C07276=1031.156,417.166,352.413,174.368,47.663,159.722
C07277=1031.145,416.920,352.461,174.356,47.658,159.719
C07278=1031.134,416.675,352.508,174.343,47.654,159.716
C07279=1031.123,416.430,352.556,174.331,47.649,159.713
C07280=1031.112,416.185,352.603,174.319,47.645,159.710
C07281=1031.101,415.939,352.650,174.306,47.640,159.707
C07282=1031.090,415.694,352.698,174.294,47.636,159.704
C07283=1031.079,415.449,352.745,174.282,47.631,159.701
C07284=1031.068,415.203,352.792,174.270,47.627,159.698
C07285=1031.057,414.958,352.839,174.258,47.622,159.696
C07286=1031.046,414.713,352.887,174.246,47.618,159.693
C07287=1031.035,414.468,352.934,174.234,47.614,159.690
C07288=1031.025,414.222,352.981,174.222,47.610,159.687
C07289=1031.014,413.977,353.028,174.210,47.605,159.684
C07290=1031.003,413.731,353.075,174.198,47.601,159.681
C07291=1030.992,413.486,353.122,174.186,47.597,159.679
C07292=1030.981,413.241,353.169,174.174,47.592,159.676
C07293=1030.970,412.995,353.216,174.162,47.588,159.673
C07294=1030.960,412.750,353.262,174.151,47.584,159.671
C07295=1030.950,412.505,353.309,174.139,47.579,159.668
C07296=1030.939,412.260,353.356,174.127,47.576,159.665
C07297=1030.928,412.014,353.403,174.115,47.571,159.662
C07298=1030.917,411.768,353.449,174.104,47.567,159.660
C07299=1030.906,411.523,353.496,174.093,47.563,159.657
C07300=1030.896,411.278,353.543,174.081,47.558,159.654
C07301=1030.885,411.032,353.589,174.070,47.554,159.652
C07302=1030.875,410.787,353.636,174.058,47.550,159.649
C07303=1030.865,410.541,353.682,174.046,47.546,159.646
C07304=1030.854,410.296,353.728,174.035,47.542,159.644
C07305=1030.843,410.051,353.775,174.024,47.538,159.641
C07306=1030.833,409.805,353.821,174.013,47.534,159.638
C07307=1030.823,409.559,353.867,174.001,47.530,159.636
C07308=1030.812,409.314,353.913,173.990,47.526,159.633
C07309=1030.800,409.049,353.962,173.978,47.522,159.630
C07310=1030.789,408.784,354.012,173.966,47.518,159.628
C07311=1030.778,408.520,354.062,173.953,47.513,159.625
C07312=1030.766,408.256,354.111,173.942,47.509,159.622
C07313=1030.756,408.010,354.158,173.930,47.505,159.620
C07314=1030.746,407.764,354.204,173.919,47.501,159.617
C07315=1030.735,407.518,354.249,173.908,47.498,159.615
C07316=1030.725,407.272,354.295,173.897,47.494,159.612
C07317=1030.715,407.028,354.340,173.886,47.490,159.610
C07318=1030.704,406.782,354.386,173.875,47.486,159.607
C07319=1030.693,406.536,354.432,173.864,47.482,159.605
C07320=1030.684,406.291,354.477,173.853,47.478,159.602
C07321=1030.673,406.045,354.523,173.843,47.475,159.600
C07322=1030.663,405.800,354.569,173.831,47.471,159.597
C07323=1030.653,405.554,354.613,173.821,47.467,159.595
C07324=1030.643,405.308,354.660,173.810,47.463,159.592
C07325=1030.633,405.062,354.705,173.799,47.460,159.590
C07326=1030.623,404.817,354.751,173.788,47.456,159.587
C07327=1030.612,404.571,354.796,173.778,47.452,159.585
C07328=1030.602,404.326,354.841,173.768,47.449,159.583
C07329=1030.593,404.080,354.886,173.756,47.445,159.580
C07330=1030.582,403.834,354.931,173.746,47.441,159.578
C07331=1030.572,403.589,354.977,173.735,47.438,159.575
C07332=1030.562,403.343,355.022,173.725,47.434,159.573
C07333=1030.552,403.098,355.067,173.714,47.430,159.571
C07334=1030.542,402.852,355.112,173.703,47.427,159.568
C07335=1030.532,402.606,355.157,173.693,47.423,159.566
C07336=1030.522,402.361,355.203,173.683,47.419,159.564
C07337=1030.512,402.116,355.247,173.673,47.416,159.561
C07338=1030.502,401.869,355.293,173.662,47.413,159.559
C07339=1030.492,401.624,355.337,173.651,47.409,159.557
C07340=1030.483,401.378,355.382,173.641,47.406,159.555
C07341=1030.473,401.131,355.427,173.631,47.402,159.552
C07342=1030.463,400.886,355.472,173.620,47.399,159.550
C07343=1030.453,400.640,355.516,173.610,47.395,159.548
C07344=1030.443,400.395,355.561,173.600,47.392,159.545
C07345=1030.433,400.150,355.605,173.590,47.388,159.543
C07346=1030.424,399.904,355.650,173.580,47.385,159.541
C07347=1030.413,399.657,355.695,173.570,47.382,159.539
C07348=1030.404,399.411,355.739,173.559,47.378,159.536
C07349=1030.394,399.166,355.784,173.549,47.375,159.534
C07350=1030.384,398.920,355.828,173.539,47.372,159.532
C07351=1030.374,398.674,355.872,173.529,47.369,159.530
C07352=1030.365,398.428,355.916,173.519,47.365,159.528
C07353=1030.354,398.183,355.960,173.509,47.361,159.525
C07354=1030.345,397.937,356.004,173.499,47.358,159.523
C07355=1030.336,397.691,356.049,173.489,47.355,159.521
C07356=1030.325,397.446,356.093,173.479,47.352,159.519
C07357=1030.316,397.199,356.137,173.469,47.349,159.517
C07358=1030.306,396.953,356.181,173.460,47.346,159.515
C07359=1030.296,396.707,356.225,173.450,47.343,159.513
C07360=1030.287,396.462,356.269,173.440,47.339,159.510
C07361=1030.278,396.217,356.313,173.430,47.336,159.508
C07362=1030.268,395.971,356.357,173.420,47.333,159.506
C07363=1030.258,395.725,356.401,173.410,47.330,159.504
C07364=1030.248,395.479,356.444,173.401,47.327,159.502
C07365=1030.239,395.233,356.488,173.391,47.324,159.500
C07366=1030.229,394.989,356.532,173.381,47.320,159.498
C07367=1030.220,394.744,356.575,173.373,47.317,159.496
C07368=1030.211,394.500,356.618,173.363,47.314,159.494
C07369=1030.201,394.255,356.662,173.353,47.312,159.492
C07370=1030.192,394.011,356.705,173.343,47.308,159.490
C07371=1030.182,393.766,356.748,173.334,47.306,159.488
C07372=1030.173,393.521,356.791,173.325,47.303,159.486
C07373=1030.164,393.275,356.835,173.315,47.299,159.484
C07374=1030.154,393.030,356.879,173.306,47.297,159.482
C07375=1030.144,392.783,356.921,173.296,47.294,159.480
C07376=1030.135,392.538,356.965,173.286,47.291,159.478
C07377=1030.125,392.291,357.008,173.278,47.288,159.476
C07378=1030.116,392.046,357.052,173.268,47.285,159.474
C07379=1030.107,391.799,357.095,173.258,47.282,159.472
C07380=1030.098,391.554,357.138,173.249,47.279,159.470
C07381=1030.088,391.308,357.181,173.240,47.276,159.468
C07382=1030.079,391.061,357.224,173.230,47.273,159.466
C07383=1030.069,390.816,357.268,173.221,47.271,159.464
C07384=1030.060,390.570,357.310,173.212,47.268,159.462
C07385=1030.051,390.323,357.353,173.203,47.265,159.460
C07386=1030.042,390.077,357.396,173.193,47.262,159.458
C07387=1030.032,389.831,357.440,173.185,47.259,159.456
C07388=1030.023,389.586,357.482,173.175,47.256,159.454
C07389=1030.013,389.339,357.525,173.166,47.254,159.452
C07390=1030.005,389.093,357.568,173.157,47.251,159.451
C07391=1029.995,388.847,357.611,173.148,47.249,159.449
C07392=1029.986,388.601,357.653,173.139,47.245,159.447
C07393=1029.976,388.355,357.696,173.130,47.243,159.445
C07394=1029.968,388.108,357.738,173.120,47.241,159.443
C07395=1029.958,387.862,357.781,173.112,47.238,159.441
C07396=1029.949,387.616,357.823,173.102,47.235,159.439
C07397=1029.941,387.370,357.866,173.094,47.232,159.438
C07398=1029.931,387.124,357.909,173.085,47.230,159.436
C07399=1029.921,386.878,357.952,173.076,47.227,159.434
C07400=1029.913,386.632,357.993,173.067,47.225,159.432
C07401=1029.903,386.386,358.036,173.059,47.222,159.430
C07402=1029.894,386.139,358.078,173.049,47.219,159.428
C07403=1029.885,385.893,358.120,173.041,47.217,159.427
C07404=1029.876,385.647,358.162,173.032,47.215,159.425
C07405=1029.866,385.401,358.204,173.023,47.212,159.423
C07406=1029.857,385.155,358.246,173.014,47.210,159.421
C07407=1029.848,384.909,358.289,173.006,47.207,159.420
C07408=1029.839,384.662,358.331,172.997,47.205,159.418
C07409=1029.830,384.415,358.372,172.988,47.202,159.416
C07410=1029.820,384.170,358.415,172.980,47.199,159.414
C07411=1029.812,383.923,358.457,172.970,47.197,159.412
C07412=1029.803,383.677,358.498,172.962,47.195,159.411
C07413=1029.794,383.431,358.540,172.954,47.192,159.409
C07414=1029.784,383.185,358.582,172.945,47.190,159.407
C07415=1029.776,382.938,358.625,172.936,47.188,159.406
C07416=1029.767,382.692,358.666,172.928,47.185,159.404
C07417=1029.758,382.445,358.708,172.919,47.183,159.402
C07418=1029.749,382.199,358.750,172.911,47.181,159.401
C07419=1029.741,381.953,358.792,172.902,47.178,159.399
C07420=1029.732,381.706,358.833,172.893,47.176,159.397
C07421=1029.723,381.460,358.875,172.885,47.174,159.395
C07422=1029.714,381.214,358.917,172.877,47.171,159.394
C07423=1029.705,380.968,358.958,172.868,47.169,159.392
C07424=1029.696,380.722,359.000,172.860,47.167,159.390
C07425=1029.688,380.495,359.038,172.852,47.165,159.389
C07426=1029.679,380.268,359.076,172.845,47.162,159.387
C07427=1029.672,380.041,359.114,172.837,47.160,159.386
C07428=1029.663,379.814,359.153,172.829,47.159,159.384
C07429=1029.656,379.587,359.191,172.822,47.156,159.383
C07430=1029.648,379.361,359.229,172.814,47.155,159.381
C07431=1029.639,379.133,359.267,172.806,47.153,159.380
C07432=1029.631,378.907,359.306,172.799,47.150,159.378
C07433=1029.623,378.660,359.347,172.790,47.148,159.377
C07434=1029.614,378.414,359.388,172.782,47.146,159.375
C07435=1029.606,378.167,359.429,172.774,47.144,159.374
C07436=1029.597,377.921,359.471,172.766,47.141,159.372
C07437=1029.589,377.675,359.512,172.758,47.140,159.370
C07438=1029.580,377.428,359.553,172.749,47.137,159.369
C07439=1029.571,377.181,359.594,172.742,47.135,159.367
C07440=1029.562,376.936,359.635,172.733,47.134,159.366
C07441=1029.554,376.689,359.676,172.725,47.132,159.364
C07442=1029.544,376.442,359.716,172.717,47.129,159.362
C07443=1029.536,376.196,359.758,172.709,47.127,159.361
C07444=1029.527,375.949,359.799,172.701,47.125,159.359
C07445=1029.519,375.703,359.839,172.693,47.123,159.358
C07446=1029.510,375.456,359.880,172.685,47.122,159.357
C07447=1029.501,375.209,359.921,172.677,47.119,159.355
C07448=1029.492,374.963,359.961,172.669,47.117,159.353
C07449=1029.484,374.717,360.003,172.661,47.115,159.352
C07450=1029.476,374.471,360.043,172.653,47.113,159.350
C07451=1029.466,374.224,360.084,172.645,47.111,159.349
C07452=1029.458,373.978,360.124,172.637,47.109,159.347
C07453=1029.450,373.731,360.165,172.629,47.108,159.346
C07454=1029.441,373.485,360.205,172.621,47.106,159.344
C07455=1029.432,373.237,360.246,172.614,47.104,159.343
C07456=1029.424,372.991,360.286,172.606,47.102,159.341
C07457=1029.416,372.745,360.326,172.598,47.100,159.340
C07458=1029.407,372.498,360.367,172.590,47.099,159.339
C07459=1029.398,372.252,360.407,172.582,47.097,159.337
C07460=1029.390,372.005,360.448,172.574,47.095,159.336
C07461=1029.382,371.758,360.488,172.566,47.093,159.334
C07462=1029.373,371.512,360.528,172.559,47.091,159.333
C07463=1029.365,371.266,360.569,172.551,47.090,159.331
C07464=1029.356,371.019,360.610,172.543,47.088,159.330
C07465=1029.348,370.772,360.649,172.536,47.085,159.328
C07466=1029.340,370.526,360.690,172.529,47.084,159.327
C07467=1029.332,370.278,360.730,172.521,47.082,159.326
C07468=1029.323,370.032,360.770,172.513,47.080,159.324
C07469=1029.315,369.786,360.811,172.505,47.079,159.323
C07470=1029.306,369.540,360.850,172.497,47.077,159.321
C07471=1029.298,369.293,360.891,172.490,47.076,159.320
C07472=1029.290,369.046,360.931,172.483,47.073,159.319
C07473=1029.282,368.799,360.970,172.475,47.072,159.317
C07474=1029.273,368.553,361.010,172.467,47.070,159.316
C07475=1029.265,368.306,361.050,172.460,47.069,159.315
C07476=1029.257,368.060,361.090,172.452,47.067,159.313
C07477=1029.248,367.812,361.129,172.444,47.066,159.312
C07478=1029.239,367.566,361.169,172.438,47.064,159.311
C07479=1029.231,367.319,361.209,172.430,47.063,159.309
C07480=1029.223,367.073,361.249,172.422,47.061,159.308
C07481=1029.214,366.826,361.288,172.415,47.059,159.306
C07482=1029.207,366.579,361.328,172.408,47.058,159.305
C07483=1029.198,366.333,361.367,172.401,47.056,159.304
C07484=1029.190,366.086,361.406,172.393,47.054,159.302
C07485=1029.182,365.870,361.442,172.386,47.053,159.301
C07486=1029.175,365.654,361.476,172.380,47.052,159.300
C07487=1029.168,365.437,361.511,172.374,47.051,159.299
C07488=1029.161,365.221,361.545,172.367,47.050,159.298
C07489=1029.154,365.004,361.580,172.361,47.048,159.297
C07490=1029.147,364.788,361.615,172.354,47.047,159.296
C07491=1029.139,364.572,361.649,172.348,47.045,159.295
C07492=1029.132,364.355,361.684,172.342,47.044,159.293
C07493=1029.124,364.109,361.723,172.334,47.043,159.292
C07494=1029.115,363.862,361.762,172.327,47.041,159.291
C07495=1029.108,363.615,361.802,172.320,47.040,159.290
C07496=1029.099,363.368,361.841,172.312,47.039,159.288
C07497=1029.091,363.121,361.880,172.306,47.037,159.287
C07498=1029.082,362.875,361.920,172.298,47.036,159.286
C07499=1029.075,362.627,361.959,172.291,47.034,159.285
C07500=1029.067,362.381,361.998,172.284,47.033,159.283
C07501=1029.059,362.135,362.037,172.276,47.031,159.282
C07502=1029.051,361.888,362.076,172.269,47.031,159.281
C07503=1029.043,361.641,362.116,172.263,47.029,159.280
C07504=1029.035,361.393,362.154,172.255,47.028,159.278
C07505=1029.026,361.147,362.194,172.248,47.026,159.277
C07506=1029.019,360.901,362.233,172.241,47.025,159.276
C07507=1029.011,360.653,362.272,172.235,47.023,159.275
C07508=1029.003,360.406,362.310,172.227,47.022,159.273
C07509=1028.994,360.160,362.350,172.220,47.021,159.272
C07510=1028.987,359.913,362.388,172.213,47.020,159.271
C07511=1028.979,359.666,362.427,172.206,47.018,159.270
C07512=1028.970,359.419,362.466,172.199,47.017,159.269
C07513=1028.962,359.172,362.504,172.192,47.016,159.268
C07514=1028.955,358.926,362.543,172.185,47.015,159.266
C07515=1028.946,358.678,362.581,172.178,47.014,159.265
C07516=1028.938,358.432,362.621,172.172,47.012,159.264
C07517=1028.930,358.185,362.659,172.164,47.012,159.263
C07518=1028.922,357.938,362.697,172.157,47.010,159.262
C07519=1028.914,357.691,362.736,172.151,47.009,159.261
C07520=1028.906,357.444,362.774,172.143,47.008,159.259
C07521=1028.898,357.197,362.813,172.137,47.007,159.258
C07522=1028.890,356.950,362.852,172.129,47.006,159.257
C07523=1028.882,356.704,362.889,172.123,47.004,159.256
C07524=1028.874,356.456,362.928,172.117,47.003,159.255
C07525=1028.866,356.210,362.966,172.109,47.003,159.254
C07526=1028.858,355.963,363.005,172.103,47.002,159.253
C07527=1028.851,355.716,363.043,172.096,47.000,159.251
C07528=1028.842,355.469,363.082,172.089,46.999,159.250
C07529=1028.835,355.222,363.120,172.082,46.998,159.249
C07530=1028.827,354.975,363.158,172.076,46.997,159.248
C07531=1028.819,354.728,363.196,172.068,46.996,159.247
C07532=1028.811,354.481,363.235,172.062,46.995,159.246
C07533=1028.803,354.235,363.272,172.056,46.994,159.245
C07534=1028.795,353.987,363.310,172.048,46.993,159.244
C07535=1028.788,353.740,363.348,172.042,46.992,159.243
C07536=1028.779,353.493,363.387,172.035,46.991,159.242
C07537=1028.771,353.246,363.424,172.029,46.990,159.241
C07538=1028.763,352.999,363.462,172.022,46.989,159.240
C07539=1028.756,352.752,363.500,172.015,46.988,159.238
C07540=1028.748,352.505,363.539,172.009,46.988,159.238
C07541=1028.740,352.258,363.576,172.002,46.987,159.236
C07542=1028.732,352.011,363.614,171.996,46.986,159.235
C07543=1028.725,351.764,363.652,171.989,46.985,159.234
C07544=1028.716,351.517,363.689,171.982,46.984,159.233
C07545=1028.710,351.303,363.722,171.977,46.983,159.232
C07546=1028.704,351.091,363.754,171.971,46.982,159.231
C07547=1028.697,350.878,363.788,171.965,46.982,159.231
C07548=1028.689,350.664,363.819,171.960,46.981,159.230
C07549=1028.683,350.452,363.852,171.954,46.981,159.229
C07550=1028.676,350.238,363.885,171.949,46.979,159.228
C07551=1028.671,350.025,363.917,171.943,46.979,159.227
C07552=1028.663,349.812,363.950,171.938,46.978,159.226
C07553=1028.656,349.565,363.987,171.931,46.977,159.225
C07554=1028.648,349.318,364.025,171.924,46.976,159.224
C07555=1028.640,349.071,364.063,171.918,46.976,159.223
C07556=1028.632,348.824,364.101,171.911,46.975,159.222
C07557=1028.620,348.434,364.159,171.901,46.974,159.221
C07558=1028.608,348.045,364.218,171.892,46.973,159.219
C07559=1028.596,347.656,364.277,171.881,46.971,159.217
C07560=1028.584,347.266,364.336,171.871,46.971,159.216
C07561=1028.576,347.020,364.373,171.865,46.970,159.215
C07562=1028.569,346.773,364.410,171.859,46.969,159.214
C07563=1028.561,346.526,364.447,171.852,46.968,159.213
C07564=1028.553,346.279,364.485,171.846,46.968,159.212
C07565=1028.545,346.032,364.522,171.839,46.967,159.211
C07566=1028.538,345.785,364.559,171.834,46.966,159.210
C07567=1028.530,345.538,364.596,171.828,46.966,159.209
C07568=1028.523,345.289,364.633,171.820,46.965,159.208
C07569=1028.515,345.042,364.670,171.814,46.965,159.207
C07570=1028.507,344.796,364.707,171.808,46.964,159.207
C07571=1028.499,344.549,364.745,171.802,46.963,159.206
C07572=1028.492,344.301,364.781,171.796,46.962,159.205
C07573=1028.485,344.054,364.819,171.789,46.962,159.204
C07574=1028.477,343.807,364.856,171.783,46.962,159.203
C07575=1028.470,343.559,364.892,171.777,46.961,159.202
C07576=1028.462,343.313,364.929,171.771,46.960,159.201
C07577=1028.454,343.066,364.966,171.765,46.960,159.200
C07578=1028.447,342.818,365.003,171.759,46.959,159.199
C07579=1028.439,342.571,365.040,171.752,46.959,159.198
C07580=1028.432,342.323,365.077,171.746,46.959,159.198
C07581=1028.424,342.077,365.113,171.740,46.958,159.196
C07582=1028.417,341.830,365.150,171.734,46.957,159.196
C07583=1028.409,341.583,365.187,171.728,46.957,159.195
C07584=1028.402,341.335,365.223,171.722,46.956,159.194
C07585=1028.394,341.088,365.260,171.716,46.956,159.193
C07586=1028.387,340.841,365.297,171.709,46.955,159.192
C07587=1028.379,340.594,365.334,171.703,46.955,159.191
C07588=1028.371,340.346,365.370,171.697,46.955,159.190
C07589=1028.364,340.099,365.407,171.691,46.954,159.190
C07590=1028.357,339.853,365.444,171.685,46.954,159.189
C07591=1028.349,339.605,365.480,171.680,46.953,159.188
C07592=1028.342,339.358,365.516,171.674,46.953,159.187
C07593=1028.334,339.110,365.552,171.668,46.953,159.186
C07594=1028.326,338.863,365.588,171.662,46.952,159.185
C07595=1028.319,338.615,365.625,171.656,46.952,159.185
C07596=1028.311,338.369,365.661,171.649,46.952,159.184
C07597=1028.304,338.121,365.698,171.643,46.951,159.183
C07598=1028.297,337.874,365.734,171.637,46.951,159.182
C07599=1028.289,337.627,365.770,171.632,46.951,159.181
C07600=1028.282,337.380,365.806,171.626,46.950,159.180
C07601=1028.274,337.132,365.843,171.620,46.950,159.180
C07602=1028.266,336.885,365.879,171.614,46.950,159.179
C07603=1028.259,336.637,365.915,171.608,46.949,159.178
C07604=1028.252,336.391,365.951,171.602,46.949,159.177
C07605=1028.244,336.103,365.993,171.595,46.949,159.176
C07606=1028.235,335.816,366.035,171.588,46.949,159.175
C07607=1028.226,335.529,366.077,171.582,46.948,159.174
C07608=1028.217,335.242,366.119,171.575,46.948,159.174
C07609=1028.211,334.995,366.155,171.569,46.947,159.173
C07610=1028.203,334.747,366.191,171.564,46.947,159.172
C07611=1028.196,334.499,366.227,171.558,46.947,159.171
C07612=1028.189,334.253,366.263,171.552,46.947,159.170
C07613=1028.181,334.005,366.299,171.546,46.947,159.170
C07614=1028.174,333.758,366.335,171.540,46.947,159.169
C07615=1028.166,333.510,366.370,171.535,46.946,159.168
C07616=1028.159,333.264,366.406,171.529,46.946,159.167
C07617=1028.151,333.016,366.442,171.523,46.946,159.167
C07618=1028.144,332.768,366.477,171.517,46.946,159.166
C07619=1028.136,332.522,366.513,171.512,46.946,159.165
C07620=1028.129,332.274,366.549,171.506,46.946,159.164
C07621=1028.122,332.027,366.585,171.500,46.946,159.164
C07622=1028.115,331.779,366.620,171.494,46.946,159.163
C07623=1028.108,331.532,366.656,171.488,46.945,159.162
C07624=1028.099,331.284,366.691,171.483,46.946,159.161
C07625=1028.092,331.038,366.727,171.477,46.946,159.161
C07626=1028.085,330.789,366.762,171.471,46.945,159.160
C07627=1028.078,330.543,366.798,171.466,46.945,159.159
C07628=1028.071,330.295,366.834,171.460,46.945,159.159
C07629=1028.064,330.048,366.869,171.454,46.946,159.158
C07630=1028.055,329.800,366.904,171.448,46.945,159.157
C07631=1028.049,329.553,366.939,171.444,46.945,159.156
C07632=1028.042,329.306,366.975,171.438,46.945,159.156
C07633=1028.034,329.058,367.011,171.432,46.945,159.155
C07634=1028.027,328.811,367.046,171.427,46.945,159.154
C07635=1028.020,328.563,367.082,171.421,46.945,159.154
C07636=1028.012,328.316,367.117,171.415,46.945,159.153
C07637=1028.005,328.069,367.152,171.410,46.945,159.152
C07638=1027.998,327.821,367.187,171.404,46.945,159.151
C07639=1027.991,327.574,367.223,171.398,46.945,159.151
C07640=1027.984,327.327,367.258,171.394,46.945,159.150
C07641=1027.976,327.079,367.293,171.388,46.945,159.149
C07642=1027.969,326.832,367.328,171.382,46.945,159.149
C07643=1027.962,326.584,367.363,171.377,46.946,159.148
C07644=1027.954,326.337,367.398,171.371,46.946,159.147
C07645=1027.946,326.090,367.432,171.366,46.946,159.147
C07646=1027.940,325.842,367.467,171.360,46.946,159.146
C07647=1027.932,325.594,367.502,171.354,46.947,159.146
C07648=1027.925,325.347,367.537,171.349,46.947,159.145
C07649=1027.917,325.099,367.571,171.343,46.947,159.144
C07650=1027.909,324.852,367.606,171.338,46.947,159.144
C07651=1027.903,324.604,367.641,171.333,46.947,159.143
C07652=1027.895,324.357,367.676,171.327,46.948,159.142
C07653=1027.888,324.110,367.711,171.322,46.948,159.142
C07654=1027.880,323.862,367.745,171.316,46.948,159.141
C07655=1027.873,323.615,367.780,171.311,46.949,159.141
C07656=1027.866,323.367,367.815,171.305,46.949,159.140
C07657=1027.859,323.120,367.849,171.301,46.949,159.139
C07658=1027.852,322.871,367.884,171.295,46.949,159.139
C07659=1027.844,322.624,367.919,171.290,46.949,159.138
C07660=1027.837,322.377,367.953,171.284,46.949,159.137
C07661=1027.831,322.160,367.983,171.280,46.950,159.137
C07662=1027.824,321.943,368.014,171.275,46.950,159.136
C07663=1027.818,321.726,368.044,171.270,46.951,159.136
C07664=1027.812,321.510,368.075,171.265,46.950,159.135
C07665=1027.806,321.292,368.105,171.261,46.951,159.135
C07666=1027.799,321.076,368.135,171.256,46.951,159.134
C07667=1027.793,320.859,368.165,171.252,46.951,159.134
C07668=1027.786,320.642,368.196,171.246,46.952,159.133
C07669=1027.779,320.394,368.230,171.242,46.952,159.133
C07670=1027.773,320.147,368.265,171.236,46.952,159.132
C07671=1027.765,319.899,368.298,171.231,46.953,159.132
C07672=1027.758,319.651,368.334,171.225,46.953,159.131
C07673=1027.751,319.404,368.368,171.220,46.953,159.130
C07674=1027.743,319.157,368.402,171.215,46.953,159.130
C07675=1027.737,318.909,368.437,171.210,46.954,159.129
C07676=1027.729,318.661,368.471,171.204,46.954,159.129
C07677=1027.722,318.414,368.505,171.199,46.955,159.128
C07678=1027.716,318.166,368.540,171.194,46.955,159.127
C07679=1027.708,317.919,368.574,171.189,46.955,159.127
C07680=1027.701,317.671,368.608,171.183,46.956,159.126
C07681=1027.695,317.424,368.642,171.178,46.956,159.126
C07682=1027.688,317.177,368.676,171.173,46.957,159.125
C07683=1027.681,316.929,368.711,171.168,46.957,159.125
C07684=1027.674,316.681,368.745,171.162,46.958,159.124
C07685=1027.666,316.434,368.779,171.158,46.957,159.124
C07686=1027.660,316.186,368.814,171.152,46.958,159.123
C07687=1027.653,315.938,368.848,171.147,46.959,159.123
C07688=1027.645,315.691,368.882,171.141,46.959,159.122
C07689=1027.639,315.443,368.916,171.137,46.959,159.121
C07690=1027.632,315.196,368.950,171.132,46.960,159.121
C07691=1027.625,314.949,368.984,171.126,46.960,159.120
C07692=1027.618,314.701,369.018,171.122,46.961,159.120
C07693=1027.611,314.454,369.053,171.116,46.962,159.119
C07694=1027.604,314.206,369.087,171.111,46.962,159.119
C07695=1027.597,313.958,369.121,171.106,46.962,159.118
C07696=1027.591,313.711,369.154,171.101,46.963,159.118
C07697=1027.583,313.463,369.188,171.096,46.964,159.117
C07698=1027.577,313.215,369.223,171.091,46.964,159.117
C07699=1027.570,312.968,369.256,171.086,46.964,159.116
C07700=1027.563,312.721,369.290,171.080,46.965,159.116
C07701=1027.557,312.473,369.324,171.076,46.965,159.115
C07702=1027.550,312.225,369.358,171.071,46.966,159.115
C07703=1027.542,311.977,369.392,171.066,46.967,159.114
C07704=1027.536,311.730,369.425,171.061,46.967,159.113
C07705=1027.529,311.482,369.460,171.055,46.967,159.113
C07706=1027.522,311.235,369.494,171.051,46.968,159.113
C07707=1027.516,310.988,369.527,171.046,46.969,159.112
C07708=1027.508,310.740,369.561,171.040,46.969,159.112
C07709=1027.501,310.492,369.595,171.036,46.970,159.111
C07710=1027.495,310.245,369.628,171.031,46.970,159.111
C07711=1027.488,309.997,369.661,171.025,46.971,159.110
C07712=1027.480,309.750,369.695,171.021,46.972,159.110
C07713=1027.473,309.502,369.728,171.016,46.973,159.109
C07714=1027.466,309.255,369.761,171.011,46.974,159.109
C07715=1027.459,309.007,369.794,171.006,46.974,159.108
C07716=1027.451,308.759,369.828,171.001,46.975,159.108
C07717=1027.445,308.512,369.861,170.996,46.976,159.107
C07718=1027.438,308.264,369.894,170.991,46.976,159.107
C07719=1027.430,308.016,369.927,170.986,46.978,159.107
C07720=1027.424,307.769,369.960,170.981,46.978,159.106
C07721=1027.417,307.554,369.989,170.977,46.979,159.106
C07722=1027.411,307.340,370.018,170.972,46.980,159.105
C07723=1027.405,307.125,370.047,170.968,46.980,159.105
C07724=1027.399,306.911,370.076,170.964,46.981,159.105
C07725=1027.393,306.696,370.103,170.960,46.982,159.104
C07726=1027.387,306.482,370.132,170.955,46.982,159.104
C07727=1027.381,306.267,370.161,170.951,46.983,159.103
C07728=1027.374,306.053,370.190,170.947,46.984,159.103
C07729=1027.368,305.805,370.223,170.943,46.984,159.103
C07730=1027.360,305.558,370.256,170.937,46.985,159.102
C07731=1027.354,305.310,370.289,170.932,46.986,159.102
C07732=1027.347,305.062,370.322,170.928,46.987,159.102
C07733=1027.340,304.814,370.356,170.923,46.988,159.101
C07734=1027.333,304.567,370.388,170.919,46.989,159.101
C07735=1027.326,304.319,370.421,170.913,46.989,159.100
C07736=1027.319,304.071,370.454,170.908,46.991,159.100
C07737=1027.312,303.824,370.487,170.904,46.991,159.099
C07738=1027.305,303.576,370.520,170.899,46.992,159.099
C07739=1027.298,303.328,370.553,170.895,46.993,159.099
C07740=1027.291,303.081,370.585,170.889,46.994,159.098
C07741=1027.284,302.833,370.619,170.884,46.995,159.098
C07742=1027.278,302.585,370.651,170.880,46.996,159.097
C07743=1027.271,302.338,370.684,170.875,46.997,159.097
C07744=1027.264,302.090,370.717,170.870,46.997,159.097
C07745=1027.258,301.842,370.749,170.865,46.999,159.096
C07746=1027.250,301.594,370.782,170.861,46.999,159.096
C07747=1027.243,301.347,370.815,170.856,47.001,159.096
C07748=1027.237,301.100,370.848,170.852,47.001,159.095
C07749=1027.229,300.852,370.881,170.847,47.002,159.095
C07750=1027.223,300.604,370.913,170.842,47.003,159.094
C07751=1027.216,300.356,370.946,170.837,47.004,159.094
C07752=1027.209,300.109,370.979,170.832,47.005,159.094
C07753=1027.203,299.861,371.011,170.828,47.006,159.093
C07754=1027.196,299.613,371.044,170.822,47.007,159.093
C07755=1027.189,299.365,371.077,170.818,47.008,159.093
C07756=1027.183,299.118,371.109,170.813,47.009,159.092
C07757=1027.176,298.870,371.142,170.809,47.010,159.092
C07758=1027.169,298.622,371.175,170.804,47.011,159.091
C07759=1027.163,298.375,371.207,170.800,47.011,159.091
C07760=1027.156,298.126,371.240,170.795,47.013,159.091
C07761=1027.149,297.879,371.273,170.791,47.014,159.090
C07762=1027.143,297.631,371.305,170.785,47.015,159.090
C07763=1027.136,297.383,371.337,170.781,47.016,159.090
C07764=1027.129,297.135,371.370,170.776,47.017,159.089
C07765=1027.122,296.888,371.403,170.772,47.018,159.089
C07766=1027.116,296.640,371.435,170.768,47.019,159.089
C07767=1027.109,296.393,371.468,170.763,47.020,159.088
C07768=1027.102,296.144,371.500,170.759,47.021,159.088
C07769=1027.096,295.896,371.533,170.753,47.022,159.088
C07770=1027.089,295.649,371.565,170.749,47.023,159.087
C07771=1027.083,295.401,371.598,170.744,47.024,159.087
C07772=1027.076,295.154,371.630,170.740,47.025,159.087
C07773=1027.069,294.905,371.662,170.735,47.026,159.086
C07774=1027.063,294.658,371.695,170.731,47.027,159.086
C07775=1027.056,294.410,371.727,170.726,47.029,159.086
C07776=1027.050,294.162,371.759,170.722,47.030,159.085
C07777=1027.043,293.915,371.791,170.717,47.030,159.085
C07778=1027.037,293.667,371.823,170.712,47.031,159.085
C07779=1027.029,293.419,371.856,170.708,47.033,159.084
C07780=1027.022,293.171,371.888,170.703,47.034,159.084
C07781=1027.012,292.760,371.941,170.696,47.036,159.084
C07782=1027.000,292.348,371.994,170.688,47.038,159.083
C07783=1026.989,291.937,372.047,170.681,47.040,159.083
C07784=1026.977,291.524,372.100,170.673,47.042,159.082
C07785=1026.971,291.276,372.132,170.669,47.043,159.082
C07786=1026.964,291.029,372.164,170.665,47.044,159.081
C07787=1026.958,290.781,372.196,170.660,47.046,159.081
C07788=1026.951,290.533,372.227,170.656,47.047,159.081
C07789=1026.944,290.285,372.258,170.651,47.049,159.081
C07790=1026.938,290.038,372.291,170.647,47.050,159.080
C07791=1026.931,289.790,372.323,170.642,47.051,159.080
C07792=1026.924,289.542,372.354,170.638,47.052,159.080
C07793=1026.917,289.293,372.386,170.633,47.054,159.080
C07794=1026.910,289.046,372.418,170.629,47.055,159.079
C07795=1026.903,288.798,372.449,170.625,47.056,159.079
C07796=1026.897,288.550,372.481,170.620,47.058,159.079
C07797=1026.891,288.302,372.513,170.616,47.059,159.079
C07798=1026.884,288.054,372.544,170.611,47.060,159.078
C07799=1026.877,287.807,372.576,170.607,47.061,159.078
C07800=1026.870,287.559,372.608,170.602,47.063,159.078
C07801=1026.863,287.311,372.639,170.598,47.064,159.078
C07802=1026.857,287.063,372.671,170.594,47.065,159.077
C07803=1026.850,286.815,372.702,170.589,47.067,159.077
C07804=1026.843,286.567,372.734,170.585,47.069,159.077
C07805=1026.836,286.319,372.765,170.580,47.070,159.077
C07806=1026.830,286.071,372.797,170.576,47.071,159.076
C07807=1026.824,285.823,372.828,170.572,47.072,159.076
C07808=1026.817,285.575,372.860,170.568,47.074,159.076
C07809=1026.810,285.328,372.891,170.564,47.075,159.076
C07810=1026.803,285.080,372.922,170.559,47.077,159.076
C07811=1026.796,284.832,372.954,170.555,47.078,159.075
C07812=1026.789,284.584,372.985,170.550,47.080,159.075
C07813=1026.783,284.335,373.016,170.546,47.081,159.075
C07814=1026.776,284.087,373.047,170.542,47.082,159.075
C07815=1026.770,283.840,373.079,170.537,47.084,159.074
C07816=1026.763,283.592,373.110,170.533,47.086,159.074
C07817=1026.756,283.345,373.141,170.528,47.088,159.074
C07818=1026.750,283.096,373.171,170.524,47.089,159.074
C07819=1026.743,282.848,373.203,170.521,47.090,159.074
C07820=1026.736,282.600,373.234,170.516,47.092,159.073
C07821=1026.729,282.353,373.266,170.512,47.093,159.073
C07822=1026.723,282.104,373.296,170.507,47.095,159.073
C07823=1026.716,281.856,373.328,170.503,47.097,159.073
C07824=1026.709,281.608,373.359,170.499,47.098,159.073
C07825=1026.702,281.361,373.390,170.494,47.100,159.072
C07826=1026.696,281.112,373.421,170.490,47.101,159.072
C07827=1026.689,280.865,373.452,170.486,47.103,159.072
C07828=1026.683,280.617,373.483,170.481,47.104,159.072
C07829=1026.676,280.368,373.514,170.478,47.106,159.072
C07830=1026.670,280.121,373.545,170.473,47.107,159.071
C07831=1026.663,279.872,373.576,170.469,47.109,159.071
C07832=1026.656,279.625,373.606,170.465,47.110,159.071
C07833=1026.650,279.377,373.638,170.460,47.112,159.071
C07834=1026.643,279.129,373.669,170.456,47.113,159.071
C07835=1026.636,278.881,373.700,170.452,47.115,159.070
C07836=1026.630,278.632,373.731,170.448,47.117,159.070
C07837=1026.619,278.233,373.781,170.441,47.119,159.070
C07838=1026.609,277.834,373.831,170.434,47.122,159.070
C07839=1026.599,277.435,373.880,170.427,47.124,159.069
C07840=1026.588,277.035,373.929,170.421,47.127,159.069
C07841=1026.581,276.787,373.960,170.417,47.129,159.069
C07842=1026.574,276.539,373.991,170.413,47.130,159.069
C07843=1026.568,276.291,374.021,170.408,47.132,159.069
C07844=1026.561,276.043,374.052,170.404,47.133,159.069
C07845=1026.554,275.795,374.083,170.400,47.135,159.068
C07846=1026.548,275.547,374.114,170.396,47.137,159.068
C07847=1026.541,275.299,374.143,170.392,47.139,159.068
C07848=1026.535,275.051,374.174,170.387,47.141,159.068
C07849=1026.528,274.803,374.205,170.384,47.143,159.068
C07850=1026.521,274.555,374.235,170.380,47.144,159.068
C07851=1026.515,274.307,374.266,170.375,47.146,159.068
C07852=1026.508,274.058,374.296,170.371,47.147,159.067
C07853=1026.501,273.811,374.327,170.367,47.149,159.067
C07854=1026.495,273.563,374.358,170.363,47.151,159.067
C07855=1026.488,273.315,374.388,170.359,47.153,159.067
C07856=1026.482,273.067,374.418,170.355,47.155,159.067
C07857=1026.475,272.818,374.448,170.350,47.157,159.067
C07858=1026.469,272.570,374.479,170.347,47.158,159.067
C07859=1026.462,272.322,374.509,170.343,47.160,159.067
C07860=1026.455,272.075,374.540,170.339,47.162,159.067
C07861=1026.448,271.826,374.570,170.334,47.163,159.066
C07862=1026.442,271.579,374.601,170.330,47.165,159.066
C07863=1026.435,271.330,374.631,170.327,47.167,159.066
C07864=1026.429,271.082,374.662,170.322,47.169,159.066
C07865=1026.422,270.834,374.691,170.318,47.170,159.066
C07866=1026.416,270.586,374.722,170.315,47.172,159.066
C07867=1026.409,270.338,374.752,170.310,47.174,159.066
C07868=1026.403,270.090,374.783,170.306,47.176,159.065
C07869=1026.396,269.842,374.812,170.303,47.178,159.066
C07870=1026.390,269.594,374.843,170.298,47.180,159.065
C07871=1026.383,269.345,374.873,170.294,47.182,159.065
C07872=1026.376,269.097,374.902,170.290,47.184,159.065
C07873=1026.370,268.849,374.933,170.286,47.186,159.065
C07874=1026.364,268.601,374.963,170.282,47.187,159.065
C07875=1026.356,268.353,374.993,170.278,47.189,159.065
C07876=1026.351,268.105,375.023,170.274,47.191,159.065
C07877=1026.343,267.857,375.053,170.270,47.194,159.065
C07878=1026.336,267.609,375.083,170.266,47.195,159.065
C07879=1026.331,267.360,375.113,170.263,47.197,159.065
C07880=1026.324,267.112,375.143,170.258,47.199,159.064
C07881=1026.317,266.865,375.173,170.254,47.201,159.064
C07882=1026.311,266.616,375.204,170.250,47.203,159.064
C07883=1026.304,266.368,375.233,170.246,47.205,159.064
C07884=1026.297,266.120,375.263,170.242,47.207,159.064
C07885=1026.291,265.872,375.293,170.238,47.209,159.064
C07886=1026.285,265.623,375.323,170.235,47.210,159.064
C07887=1026.278,265.376,375.352,170.230,47.213,159.064
C07888=1026.271,265.128,375.382,170.227,47.215,159.064
C07889=1026.265,264.879,375.412,170.223,47.217,159.064
C07890=1026.258,264.632,375.441,170.218,47.219,159.064
C07891=1026.251,264.384,375.471,170.215,47.221,159.064
C07892=1026.245,264.135,375.501,170.211,47.223,159.064
C07893=1026.235,263.740,375.548,170.204,47.226,159.064
C07894=1026.224,263.346,375.596,170.198,47.229,159.063
C07895=1026.214,262.951,375.643,170.192,47.233,159.063
C07896=1026.203,262.555,375.690,170.186,47.236,159.063
C07897=1026.197,262.308,375.720,170.182,47.238,159.063
C07898=1026.190,262.060,375.749,170.178,47.240,159.063
C07899=1026.183,261.812,375.779,170.174,47.242,159.063
C07900=1026.178,261.563,375.809,170.171,47.244,159.063
C07901=1026.170,261.315,375.839,170.166,47.246,159.063
C07902=1026.164,261.067,375.868,170.163,47.248,159.063
C07903=1026.158,260.819,375.897,170.159,47.251,159.063
C07904=1026.151,260.570,375.927,170.155,47.252,159.063
C07905=1026.145,260.322,375.956,170.151,47.255,159.063
C07906=1026.138,260.074,375.984,170.147,47.257,159.063
C07907=1026.130,259.826,376.015,170.144,47.259,159.063
C07908=1026.124,259.578,376.044,170.139,47.262,159.063
C07909=1026.117,259.329,376.073,170.136,47.263,159.063
C07910=1026.111,259.081,376.102,170.132,47.266,159.063
C07911=1026.104,258.833,376.130,170.127,47.268,159.063
C07912=1026.097,258.585,376.161,170.124,47.270,159.063
C07913=1026.091,258.337,376.190,170.121,47.273,159.063
C07914=1026.084,258.089,376.219,170.116,47.275,159.063
C07915=1026.077,257.840,376.247,170.112,47.277,159.063
C07916=1026.071,257.592,376.277,170.109,47.279,159.063
C07917=1026.064,257.343,376.306,170.105,47.281,159.063
C07918=1026.057,257.095,376.335,170.101,47.284,159.063
C07919=1026.050,256.847,376.363,170.097,47.286,159.063
C07920=1026.044,256.600,376.393,170.094,47.288,159.063
C07921=1026.037,256.351,376.423,170.089,47.291,159.063
C07922=1026.031,256.103,376.452,170.086,47.293,159.063
C07923=1026.024,255.855,376.480,170.082,47.295,159.063
C07924=1026.017,255.606,376.509,170.079,47.297,159.063
C07925=1026.011,255.358,376.539,170.074,47.300,159.063
C07926=1026.004,255.110,376.568,170.071,47.302,159.063
C07927=1025.997,254.862,376.596,170.067,47.305,159.063
C07928=1025.991,254.613,376.625,170.063,47.307,159.063
C07929=1025.984,254.365,376.654,170.059,47.309,159.063
C07930=1025.978,254.117,376.684,170.056,47.311,159.063
C07931=1025.971,253.869,376.712,170.052,47.314,159.063
C07932=1025.964,253.620,376.741,170.048,47.316,159.063
C07933=1025.958,253.372,376.770,170.044,47.318,159.063
C07934=1025.952,253.124,376.799,170.041,47.321,159.063
C07935=1025.945,252.876,376.827,170.037,47.323,159.063
C07936=1025.938,252.627,376.857,170.033,47.326,159.063
C07937=1025.932,252.379,376.886,170.029,47.327,159.063
C07938=1025.926,252.131,376.915,170.026,47.330,159.063
C07939=1025.919,251.883,376.943,170.022,47.332,159.063
C07940=1025.913,251.635,376.972,170.018,47.335,159.063
C07941=1025.906,251.387,377.001,170.014,47.337,159.064
C07942=1025.899,251.138,377.031,170.011,47.340,159.064
C07943=1025.893,250.889,377.058,170.007,47.341,159.064
C07944=1025.887,250.641,377.087,170.004,47.344,159.064
C07945=1025.880,250.393,377.116,169.999,47.347,159.064
C07946=1025.874,250.145,377.145,169.996,47.349,159.064
C07947=1025.867,249.897,377.174,169.993,47.351,159.064
C07948=1025.861,249.648,377.202,169.989,47.354,159.064
C07949=1025.851,249.252,377.249,169.983,47.358,159.064
C07950=1025.840,248.855,377.295,169.977,47.361,159.064
C07951=1025.830,248.459,377.341,169.971,47.365,159.064
C07952=1025.819,248.063,377.386,169.966,47.369,159.064
C07953=1025.813,247.814,377.415,169.962,47.371,159.064
C07954=1025.807,247.566,377.444,169.958,47.374,159.064
C07955=1025.801,247.318,377.473,169.954,47.376,159.064
C07956=1025.794,247.070,377.501,169.951,47.379,159.064
C07957=1025.788,246.822,377.530,169.947,47.381,159.064
C07958=1025.781,246.573,377.559,169.944,47.384,159.065
C07959=1025.775,246.325,377.586,169.940,47.386,159.065
C07960=1025.768,246.077,377.615,169.936,47.389,159.065
C07961=1025.763,245.828,377.644,169.933,47.391,159.065
C07962=1025.756,245.580,377.673,169.929,47.394,159.065
C07963=1025.749,245.332,377.701,169.926,47.396,159.065
C07964=1025.743,245.083,377.730,169.923,47.398,159.065
C07965=1025.737,244.835,377.759,169.918,47.401,159.065
C07966=1025.730,244.587,377.786,169.915,47.403,159.065
C07967=1025.724,244.339,377.815,169.911,47.406,159.065
C07968=1025.718,244.090,377.844,169.908,47.408,159.065
C07969=1025.711,243.842,377.872,169.904,47.411,159.065
C07970=1025.705,243.593,377.900,169.900,47.413,159.065
C07971=1025.698,243.346,377.929,169.897,47.416,159.065
C07972=1025.692,243.097,377.957,169.893,47.418,159.065
C07973=1025.685,242.849,377.986,169.890,47.420,159.065
C07974=1025.679,242.600,378.014,169.887,47.424,159.066
C07975=1025.673,242.352,378.042,169.882,47.426,159.066
C07976=1025.667,242.104,378.071,169.879,47.429,159.066
C07977=1025.660,241.855,378.098,169.875,47.431,159.066
C07978=1025.653,241.607,378.126,169.872,47.433,159.066
C07979=1025.647,241.359,378.155,169.869,47.437,159.066
C07980=1025.641,241.111,378.183,169.864,47.439,159.066
C07981=1025.635,240.862,378.211,169.861,47.442,159.066
C07982=1025.628,240.614,378.239,169.857,47.444,159.066
C07983=1025.622,240.366,378.268,169.854,47.447,159.067
C07984=1025.615,240.117,378.295,169.851,47.449,159.067
C07985=1025.609,239.869,378.323,169.846,47.452,159.067
C07986=1025.602,239.621,378.352,169.843,47.455,159.067
C07987=1025.596,239.372,378.380,169.840,47.458,159.067
C07988=1025.589,239.124,378.408,169.837,47.460,159.067
C07989=1025.582,238.875,378.435,169.833,47.463,159.067
C07990=1025.576,238.627,378.463,169.829,47.466,159.067
C07991=1025.570,238.378,378.491,169.826,47.468,159.067
C07992=1025.564,238.130,378.519,169.822,47.471,159.068
C07993=1025.557,237.882,378.547,169.819,47.474,159.068
C07994=1025.550,237.634,378.575,169.815,47.476,159.068
C07995=1025.543,237.386,378.603,169.811,47.479,159.068
C07996=1025.537,237.137,378.630,169.808,47.482,159.068
C07997=1025.531,236.888,378.659,169.805,47.485,159.068
C07998=1025.524,236.640,378.686,169.802,47.487,159.068
C07999=1025.517,236.391,378.714,169.797,47.491,159.069
C08000=1025.511,236.143,378.742,169.794,47.493,159.069
C08001=1025.504,235.895,378.769,169.791,47.496,159.069
C08002=1025.498,235.647,378.797,169.787,47.499,159.069
C08003=1025.491,235.398,378.825,169.784,47.502,159.069
C08004=1025.484,235.150,378.853,169.780,47.504,159.069
C08005=1025.474,234.748,378.897,169.775,47.509,159.070
C08006=1025.464,234.345,378.942,169.769,47.513,159.070
C08007=1025.453,233.942,378.987,169.763,47.518,159.070
C08008=1025.442,233.540,379.032,169.758,47.522,159.070
C08009=1025.436,233.291,379.060,169.755,47.525,159.070
C08010=1025.431,233.043,379.087,169.751,47.528,159.071
C08011=1025.424,232.794,379.115,169.748,47.531,159.071
C08012=1025.417,232.546,379.142,169.744,47.534,159.071
C08013=1025.411,232.298,379.170,169.740,47.537,159.071
C08014=1025.405,232.051,379.198,169.737,47.540,159.071
C08015=1025.397,231.803,379.225,169.734,47.542,159.071
C08016=1025.391,231.555,379.252,169.731,47.545,159.072
C08017=1025.385,231.307,379.280,169.726,47.548,159.072
C08018=1025.379,231.060,379.307,169.723,47.551,159.072
C08019=1025.372,230.811,379.335,169.720,47.554,159.072
C08020=1025.365,230.565,379.362,169.717,47.556,159.072
C08021=1025.360,230.316,379.389,169.714,47.559,159.072
C08022=1025.353,230.068,379.417,169.711,47.562,159.073
C08023=1025.346,229.819,379.444,169.706,47.565,159.073
C08024=1025.340,229.570,379.471,169.703,47.568,159.073
C08025=1025.334,229.322,379.499,169.700,47.571,159.073
C08026=1025.327,229.074,379.526,169.696,47.574,159.073
C08027=1025.321,228.825,379.553,169.693,47.577,159.073
C08028=1025.314,228.577,379.581,169.689,47.580,159.074
C08029=1025.308,228.329,379.609,169.686,47.583,159.074
C08030=1025.302,228.080,379.636,169.683,47.586,159.074
C08031=1025.295,227.831,379.663,169.680,47.589,159.074
C08032=1025.289,227.583,379.690,169.677,47.592,159.074
C08033=1025.282,227.334,379.718,169.672,47.595,159.074
C08034=1025.275,227.086,379.745,169.669,47.598,159.075
C08035=1025.269,226.838,379.771,169.666,47.601,159.075
C08036=1025.263,226.590,379.799,169.663,47.604,159.075
C08037=1025.256,226.340,379.826,169.660,47.607,159.075
C08038=1025.249,226.093,379.853,169.656,47.610,159.076
C08039=1025.243,225.844,379.880,169.652,47.613,159.076
C08040=1025.237,225.595,379.907,169.649,47.616,159.076
C08041=1025.230,225.348,379.934,169.646,47.619,159.076
C08042=1025.223,225.098,379.961,169.642,47.622,159.076
C08043=1025.217,224.850,379.989,169.639,47.625,159.077
C08044=1025.210,224.602,380.015,169.636,47.628,159.077
C08045=1025.204,224.353,380.042,169.633,47.631,159.077
C08046=1025.197,224.104,380.069,169.629,47.634,159.077
C08047=1025.191,223.856,380.096,169.625,47.638,159.078
C08048=1025.184,223.608,380.123,169.622,47.641,159.078
C08049=1025.178,223.359,380.150,169.619,47.644,159.078
C08050=1025.172,223.111,380.177,169.616,47.647,159.078
C08051=1025.164,222.862,380.204,169.613,47.650,159.079
C08052=1025.159,222.614,380.231,169.609,47.654,159.079
C08053=1025.152,222.365,380.258,169.606,47.657,159.079
C08054=1025.145,222.117,380.285,169.603,47.660,159.079
C08055=1025.139,221.869,380.311,169.599,47.663,159.079
C08056=1025.133,221.619,380.338,169.596,47.665,159.079
C08057=1025.126,221.372,380.365,169.592,47.669,159.080
C08058=1025.119,221.123,380.392,169.589,47.672,159.080
C08059=1025.114,220.875,380.419,169.586,47.675,159.080
C08060=1025.107,220.626,380.445,169.583,47.678,159.080
C08061=1025.096,220.214,380.490,169.577,47.683,159.081
C08062=1025.086,219.803,380.535,169.572,47.688,159.081
C08063=1025.075,219.391,380.579,169.566,47.694,159.082
C08064=1025.064,218.979,380.624,169.561,47.699,159.082
C08065=1025.058,218.731,380.650,169.558,47.703,159.082
C08066=1025.052,218.482,380.677,169.555,47.706,159.083
C08067=1025.045,218.234,380.703,169.551,47.709,159.083
C08068=1025.038,217.985,380.730,169.548,47.712,159.083
C08069=1025.032,217.737,380.756,169.544,47.715,159.083
C08070=1025.025,217.488,380.783,169.541,47.718,159.084
C08071=1025.019,217.240,380.810,169.538,47.722,159.084
C08072=1025.012,216.991,380.836,169.534,47.725,159.084
C08073=1025.005,216.743,380.862,169.531,47.728,159.084
C08074=1024.999,216.494,380.889,169.528,47.732,159.085
C08075=1024.992,216.246,380.915,169.525,47.735,159.085
C08076=1024.986,215.997,380.942,169.521,47.739,159.085
C08077=1024.980,215.749,380.968,169.518,47.742,159.085
C08078=1024.972,215.500,380.995,169.515,47.745,159.086
C08079=1024.967,215.252,381.021,169.512,47.748,159.086
C08080=1024.960,215.003,381.048,169.508,47.752,159.086
C08081=1024.954,214.755,381.074,169.505,47.755,159.087
C08082=1024.947,214.505,381.100,169.502,47.758,159.087
C08083=1024.940,214.257,381.126,169.499,47.761,159.087
C08084=1024.934,214.008,381.153,169.496,47.765,159.087
C08085=1024.928,213.760,381.179,169.492,47.768,159.088
C08086=1024.922,213.512,381.206,169.489,47.772,159.088
C08087=1024.915,213.263,381.232,169.486,47.775,159.088
C08088=1024.908,213.015,381.258,169.483,47.778,159.089
C08089=1024.902,212.766,381.285,169.480,47.782,159.089
C08090=1024.895,212.518,381.311,169.476,47.785,159.089
C08091=1024.888,212.269,381.337,169.473,47.789,159.089
C08092=1024.883,212.020,381.364,169.470,47.792,159.090
C08093=1024.876,211.772,381.390,169.467,47.795,159.090
C08094=1024.870,211.523,381.417,169.464,47.799,159.090
C08095=1024.863,211.275,381.443,169.460,47.802,159.090
C08096=1024.856,211.026,381.469,169.457,47.805,159.091
C08097=1024.851,210.777,381.495,169.454,47.809,159.091
C08098=1024.844,210.529,381.521,169.451,47.812,159.091
C08099=1024.837,210.280,381.548,169.448,47.815,159.092
C08100=1024.831,210.032,381.574,169.444,47.819,159.092
C08101=1024.825,209.783,381.600,169.441,47.822,159.092
C08102=1024.818,209.535,381.626,169.438,47.826,159.093
C08103=1024.811,209.287,381.652,169.435,47.829,159.093
C08104=1024.805,209.039,381.678,169.433,47.833,159.093
C08105=1024.798,208.789,381.704,169.428,47.836,159.093
C08106=1024.792,208.541,381.730,169.426,47.840,159.094
C08107=1024.786,208.293,381.757,169.423,47.843,159.094
C08108=1024.779,208.043,381.782,169.420,47.847,159.095
C08109=1024.773,207.795,381.808,169.416,47.850,159.095
C08110=1024.766,207.546,381.834,169.413,47.854,159.095
C08111=1024.759,207.298,381.860,169.410,47.857,159.095
C08112=1024.753,207.050,381.887,169.407,47.861,159.096
C08113=1024.747,206.801,381.912,169.404,47.864,159.096
C08114=1024.740,206.552,381.938,169.400,47.868,159.096
C08115=1024.734,206.304,381.964,169.397,47.871,159.097
C08116=1024.727,206.056,381.990,169.394,47.875,159.097
C08117=1024.716,205.647,382.033,169.389,47.881,159.098
C08118=1024.706,205.239,382.074,169.384,47.887,159.098
C08119=1024.695,204.832,382.117,169.379,47.893,159.099
C08120=1024.684,204.424,382.159,169.374,47.899,159.099
C08121=1024.660,203.392,382.260,168.969,47.798,159.023
C08122=1024.655,203.143,382.284,168.965,47.803,159.023
C08123=1024.649,202.894,382.309,168.961,47.807,159.024
C08124=1024.643,202.646,382.333,168.956,47.811,159.024
C08125=1024.637,202.397,382.357,168.953,47.816,159.025
C08126=1024.632,202.148,382.382,168.949,47.820,159.025
C08127=1024.626,201.900,382.406,168.944,47.824,159.025
C08128=1024.621,201.650,382.431,168.940,47.829,159.026
C08129=1024.614,201.402,382.454,168.936,47.833,159.026
C08130=1024.609,201.154,382.478,168.932,47.838,159.026
C08131=1024.603,200.904,382.503,168.928,47.842,159.027
C08132=1024.598,200.656,382.527,168.923,47.846,159.027
C08133=1024.592,200.407,382.550,168.920,47.851,159.027
C08134=1024.586,200.157,382.575,168.916,47.855,159.028
C08135=1024.581,199.909,382.599,168.912,47.860,159.028
C08136=1024.575,199.661,382.623,168.908,47.864,159.028
C08137=1024.569,199.411,382.647,168.903,47.869,159.029
C08138=1024.563,199.163,382.671,168.900,47.874,159.029
C08139=1024.558,198.914,382.695,168.896,47.878,159.030
C08140=1024.551,198.665,382.719,168.892,47.883,159.030
C08141=1024.545,198.417,382.742,168.888,47.887,159.030
C08142=1024.540,198.167,382.766,168.883,47.892,159.031
C08143=1024.534,197.919,382.790,168.880,47.897,159.031
C08144=1024.529,197.670,382.814,168.876,47.901,159.032
C08145=1024.522,197.422,382.838,168.871,47.906,159.032
C08146=1024.517,197.172,382.861,168.868,47.910,159.032
C08147=1024.511,196.923,382.885,168.863,47.915,159.033
C08148=1024.505,196.675,382.909,168.860,47.920,159.033
C08149=1024.500,196.426,382.933,168.856,47.924,159.034
C08150=1024.494,196.178,382.956,168.851,47.929,159.034
C08151=1024.488,195.928,382.980,168.848,47.934,159.035
C08152=1024.482,195.679,383.004,168.844,47.938,159.035
C08153=1024.476,195.431,383.027,168.840,47.943,159.035
C08154=1024.471,195.182,383.051,168.836,47.947,159.036
C08155=1024.465,194.934,383.075,168.831,47.952,159.036
C08156=1024.459,194.684,383.099,168.828,47.957,159.037
C08157=1024.453,194.435,383.122,168.824,47.961,159.037
C08158=1024.448,194.187,383.145,168.819,47.966,159.037
C08159=1024.442,193.938,383.169,168.816,47.970,159.038
C08160=1024.437,193.689,383.192,168.812,47.974,159.038
C08161=1024.430,193.440,383.216,168.809,47.979,159.039
C08162=1024.425,193.191,383.240,168.804,47.984,159.039
C08163=1024.419,192.943,383.264,168.800,47.988,159.039
C08164=1024.414,192.693,383.287,168.797,47.993,159.040
C08165=1024.408,192.445,383.311,168.792,47.998,159.040
C08166=1024.402,192.196,383.334,168.789,48.002,159.041
C08167=1024.397,191.948,383.358,168.785,48.007,159.041
C08168=1024.391,191.698,383.381,168.781,48.012,159.041
C08169=1024.385,191.449,383.406,168.777,48.016,159.042
C08170=1024.380,191.201,383.429,168.773,48.021,159.042
C08171=1024.374,190.952,383.452,168.770,48.026,159.043
C08172=1024.369,190.703,383.476,168.765,48.030,159.043
C08173=1024.363,190.454,383.499,168.762,48.035,159.043
C08174=1024.357,190.206,383.522,168.758,48.040,159.044
C08175=1024.352,189.957,383.546,168.755,48.044,159.044
C08176=1024.346,189.708,383.569,168.750,48.049,159.045
C08177=1024.341,189.459,383.593,168.746,48.053,159.045
C08178=1024.335,189.210,383.616,168.743,48.058,159.046
C08179=1024.329,188.961,383.639,168.739,48.062,159.046
C08180=1024.324,188.713,383.663,168.735,48.067,159.046
C08181=1024.318,188.464,383.686,168.731,48.072,159.047
C08182=1024.311,188.181,383.713,168.727,48.077,159.047
C08183=1024.306,187.899,383.740,168.722,48.082,159.048
C08184=1024.299,187.616,383.766,168.718,48.088,159.048
C08185=1024.293,187.334,383.792,168.713,48.093,159.049
C08186=1024.287,187.086,383.815,168.710,48.098,159.049
C08187=1024.282,186.837,383.839,168.706,48.102,159.050
C08188=1024.276,186.588,383.862,168.703,48.107,159.050
C08189=1024.270,186.339,383.885,168.699,48.111,159.051
C08190=1024.265,186.090,383.909,168.696,48.116,159.051
C08191=1024.259,185.842,383.933,168.691,48.120,159.051
C08192=1024.254,185.592,383.956,168.688,48.125,159.052
C08193=1024.249,185.344,383.979,168.684,48.130,159.052
C08194=1024.243,185.095,384.002,168.680,48.134,159.053
C08195=1024.238,184.845,384.026,168.677,48.139,159.053
C08196=1024.232,184.597,384.049,168.673,48.144,159.053
C08197=1024.226,184.348,384.072,168.669,48.149,159.054
C08198=1024.221,184.099,384.096,168.665,48.153,159.054
C08199=1024.215,183.850,384.119,168.662,48.158,159.055
C08200=1024.210,183.601,384.142,168.658,48.162,159.055
C08201=1024.205,183.353,384.165,168.655,48.167,159.056
C08202=1024.200,183.104,384.188,168.651,48.171,159.056
C08203=1024.194,182.855,384.211,168.647,48.176,159.056
C08204=1024.189,182.606,384.234,168.644,48.181,159.057
C08205=1024.183,182.357,384.257,168.639,48.186,159.057
C08206=1024.177,182.108,384.280,168.636,48.191,159.058
C08207=1024.171,181.859,384.302,168.633,48.195,159.058
C08208=1024.165,181.611,384.325,168.629,48.200,159.059
C08209=1024.160,181.361,384.348,168.625,48.205,159.059
C08210=1024.154,181.112,384.371,168.621,48.210,159.060
C08211=1024.148,180.864,384.393,168.618,48.215,159.060
C08212=1024.142,180.615,384.416,168.614,48.220,159.061
C08213=1024.136,180.365,384.438,168.610,48.225,159.061
C08214=1024.131,180.116,384.461,168.606,48.230,159.062
C08215=1024.124,179.868,384.483,168.603,48.234,159.062
C08216=1024.119,179.619,384.506,168.599,48.239,159.063
C08217=1024.113,179.369,384.529,168.595,48.244,159.063
C08218=1024.107,179.121,384.551,168.591,48.249,159.063
C08219=1024.101,178.872,384.574,168.588,48.254,159.064
C08220=1024.096,178.624,384.596,168.585,48.259,159.064
C08221=1024.090,178.374,384.619,168.581,48.264,159.065
C08222=1024.084,178.125,384.641,168.577,48.269,159.066
C08223=1024.078,177.877,384.664,168.573,48.274,159.066
C08224=1024.073,177.627,384.686,168.570,48.279,159.066
C08225=1024.067,177.378,384.709,168.567,48.284,159.067
C08226=1024.061,177.130,384.730,168.563,48.288,159.067
C08227=1024.056,176.881,384.753,168.560,48.293,159.068
C08228=1024.050,176.632,384.776,168.555,48.298,159.068
C08229=1024.044,176.383,384.798,168.552,48.303,159.069
C08230=1024.038,176.134,384.821,168.548,48.308,159.069
C08231=1024.033,175.886,384.843,168.545,48.313,159.070
C08232=1024.028,175.636,384.866,168.541,48.317,159.070
C08233=1024.021,175.387,384.888,168.538,48.322,159.071
C08234=1024.016,175.138,384.910,168.534,48.328,159.071
C08235=1024.010,174.889,384.933,168.530,48.333,159.072
C08236=1024.004,174.641,384.955,168.527,48.338,159.072
C08237=1023.999,174.392,384.977,168.523,48.342,159.073
C08238=1023.993,174.142,385.000,168.520,48.347,159.073
C08239=1023.987,173.894,385.022,168.517,48.352,159.074
C08240=1023.981,173.644,385.044,168.513,48.357,159.074
C08241=1023.976,173.396,385.067,168.510,48.362,159.075
C08242=1023.971,173.146,385.089,168.505,48.367,159.075
C08243=1023.964,172.898,385.111,168.502,48.372,159.076
C08244=1023.959,172.649,385.133,168.498,48.376,159.076
C08245=1023.954,172.400,385.156,168.495,48.381,159.077
C08246=1023.946,172.117,385.182,168.491,48.387,159.077
C08247=1023.941,171.834,385.207,168.488,48.392,159.078
C08248=1023.935,171.552,385.232,168.483,48.398,159.078
C08249=1023.928,171.268,385.257,168.479,48.404,159.079
C08250=1023.923,171.020,385.280,168.476,48.409,159.079
C08251=1023.917,170.771,385.302,168.472,48.414,159.080
C08252=1023.911,170.522,385.324,168.469,48.418,159.080
C08253=1023.906,170.273,385.346,168.466,48.423,159.081
C08254=1023.900,170.024,385.368,168.462,48.428,159.081
C08255=1023.894,169.775,385.391,168.459,48.433,159.082
C08256=1023.889,169.526,385.412,168.455,48.438,159.082
C08257=1023.884,169.277,385.435,168.452,48.443,159.083
C08258=1023.877,169.028,385.457,168.447,48.448,159.083
C08259=1023.872,168.779,385.479,168.444,48.452,159.084
C08260=1023.867,168.530,385.501,168.441,48.458,159.084
C08261=1023.860,168.281,385.523,168.437,48.463,159.085
C08262=1023.856,168.032,385.545,168.434,48.468,159.085
C08263=1023.850,167.783,385.568,168.431,48.472,159.086
C08264=1023.844,167.535,385.590,168.427,48.477,159.086
C08265=1023.839,167.286,385.612,168.424,48.482,159.087
C08266=1023.834,167.036,385.634,168.420,48.487,159.087
C08267=1023.828,166.788,385.656,168.417,48.492,159.088
C08268=1023.822,166.539,385.678,168.413,48.497,159.088
C08269=1023.817,166.290,385.700,168.410,48.501,159.089
C08270=1023.811,166.041,385.722,168.406,48.506,159.089
C08271=1023.806,165.792,385.745,168.403,48.512,159.090
C08272=1023.801,165.543,385.767,168.400,48.517,159.090
C08273=1023.795,165.294,385.788,168.396,48.521,159.091
C08274=1023.790,165.045,385.810,168.393,48.526,159.091
C08275=1023.784,164.795,385.832,168.390,48.531,159.092
C08276=1023.778,164.547,385.854,168.386,48.536,159.092
C08277=1023.773,164.298,385.876,168.383,48.541,159.093
C08278=1023.768,164.049,385.898,168.380,48.545,159.093
C08279=1023.762,163.800,385.920,168.377,48.550,159.094
C08280=1023.757,163.551,385.942,168.373,48.555,159.094
C08281=1023.752,163.302,385.964,168.370,48.560,159.095
C08282=1023.746,163.054,385.986,168.367,48.565,159.095
C08283=1023.740,162.804,386.008,168.364,48.570,159.096
C08284=1023.736,162.555,386.030,168.360,48.575,159.096
C08285=1023.729,162.306,386.052,168.357,48.580,159.097
C08286=1023.725,162.057,386.074,168.353,48.585,159.097
C08287=1023.719,161.808,386.096,168.350,48.589,159.098
C08288=1023.714,161.559,386.117,168.346,48.594,159.098
C08289=1023.708,161.310,386.139,168.343,48.599,159.099
C08290=1023.703,161.061,386.161,168.340,48.604,159.099
C08291=1023.697,160.812,386.183,168.336,48.609,159.100
C08292=1023.692,160.564,386.205,168.334,48.613,159.100
C08293=1023.687,160.314,386.228,168.330,48.618,159.101
C08294=1023.681,160.066,386.249,168.327,48.623,159.101
C08295=1023.676,159.817,386.271,168.324,48.629,159.102
C08296=1023.671,159.567,386.293,168.320,48.633,159.102
C08297=1023.665,159.319,386.314,168.317,48.638,159.103
C08298=1023.660,159.069,386.337,168.314,48.643,159.103
C08299=1023.654,158.821,386.358,168.310,48.648,159.104
C08300=1023.648,158.571,386.379,168.307,48.653,159.104
C08301=1023.643,158.322,386.400,168.304,48.658,159.105
C08302=1023.637,158.073,386.422,168.300,48.663,159.105
C08303=1023.632,157.824,386.444,168.297,48.668,159.106
C08304=1023.626,157.575,386.465,168.294,48.674,159.106
C08305=1023.621,157.326,386.486,168.290,48.678,159.107
C08306=1023.616,157.077,386.508,168.287,48.683,159.107
C08307=1023.610,156.828,386.529,168.284,48.689,159.108
C08308=1023.604,156.580,386.550,168.280,48.694,159.109
C08309=1023.598,156.330,386.571,168.277,48.699,159.109
C08310=1023.592,156.047,386.596,168.274,48.704,159.110
C08311=1023.585,155.764,386.620,168.270,48.710,159.110
C08312=1023.580,155.481,386.644,168.267,48.716,159.111
C08313=1023.573,155.197,386.669,168.263,48.721,159.111
C08314=1023.567,154.949,386.690,168.260,48.727,159.112
C08315=1023.562,154.700,386.711,168.256,48.732,159.113
C08316=1023.556,154.450,386.733,168.253,48.737,159.113
C08317=1023.550,154.202,386.754,168.250,48.742,159.114
C08318=1023.545,153.952,386.775,168.246,48.747,159.114
C08319=1023.540,153.703,386.797,168.243,48.752,159.115
C08320=1023.534,153.455,386.818,168.240,48.757,159.115
C08321=1023.528,153.205,386.839,168.237,48.762,159.116
C08322=1023.523,152.956,386.860,168.234,48.767,159.116
C08323=1023.517,152.707,386.881,168.231,48.772,159.117
C08324=1023.511,152.458,386.902,168.227,48.777,159.118
C08325=1023.506,152.210,386.923,168.224,48.782,159.118
C08326=1023.500,151.960,386.944,168.221,48.788,159.119
C08327=1023.494,151.711,386.966,168.218,48.793,159.119
C08328=1023.490,151.462,386.987,168.214,48.798,159.120
C08329=1023.484,151.213,387.008,168.211,48.803,159.120
C08330=1023.478,150.963,387.029,168.208,48.808,159.121
C08331=1023.473,150.715,387.050,168.205,48.813,159.121
C08332=1023.467,150.465,387.071,168.201,48.818,159.122
C08333=1023.461,150.217,387.092,168.198,48.823,159.122
C08334=1023.456,149.968,387.113,168.196,48.828,159.123
C08335=1023.450,149.718,387.135,168.192,48.833,159.124
C08336=1023.445,149.469,387.155,168.189,48.838,159.124
C08337=1023.439,149.221,387.176,168.186,48.844,159.125
C08338=1023.434,148.972,387.197,168.182,48.849,159.125
C08339=1023.428,148.722,387.218,168.179,48.854,159.126
C08340=1023.422,148.473,387.239,168.176,48.859,159.126
C08341=1023.417,148.224,387.260,168.173,48.864,159.127
C08342=1023.411,147.975,387.281,168.170,48.870,159.127
C08343=1023.406,147.726,387.302,168.167,48.874,159.128
C08344=1023.400,147.477,387.323,168.164,48.879,159.128
C08345=1023.395,147.228,387.344,168.161,48.885,159.129
C08346=1023.389,146.978,387.365,168.157,48.889,159.130
C08347=1023.384,146.730,387.386,168.154,48.895,159.130
C08348=1023.378,146.481,387.407,168.151,48.900,159.131
C08349=1023.372,146.232,387.426,168.147,48.905,159.131
C08350=1023.366,145.983,387.448,168.144,48.910,159.132
C08351=1023.361,145.734,387.469,168.142,48.915,159.132
C08352=1023.356,145.484,387.489,168.139,48.921,159.133
C08353=1023.350,145.235,387.510,168.136,48.925,159.133
C08354=1023.344,144.986,387.531,168.133,48.931,159.134
C08355=1023.338,144.737,387.551,168.129,48.936,159.135
C08356=1023.333,144.488,387.572,168.126,48.941,159.135
C08357=1023.328,144.239,387.592,168.123,48.946,159.136
C08358=1023.322,143.989,387.613,168.120,48.952,159.136
C08359=1023.316,143.741,387.634,168.116,48.957,159.137
C08360=1023.310,143.492,387.655,168.114,48.962,159.138
C08361=1023.305,143.243,387.675,168.111,48.967,159.138
C08362=1023.300,142.994,387.696,168.108,48.973,159.139
C08363=1023.293,142.744,387.716,168.104,48.977,159.139
C08364=1023.288,142.495,387.737,168.101,48.982,159.140
C08365=1023.282,142.246,387.758,168.098,48.988,159.140
C08366=1023.277,141.997,387.778,168.095,48.993,159.141
C08367=1023.271,141.749,387.798,168.092,48.998,159.141
C08368=1023.265,141.499,387.819,168.089,49.003,159.142
C08369=1023.260,141.250,387.840,168.086,49.009,159.143
C08370=1023.255,141.000,387.860,168.083,49.013,159.143
C08371=1023.249,140.752,387.880,168.080,49.019,159.144
C08372=1023.243,140.503,387.901,168.076,49.024,159.144
C08373=1023.238,140.254,387.922,168.073,49.030,159.145
C08374=1023.232,139.970,387.945,168.070,49.035,159.146
C08375=1023.225,139.686,387.969,168.066,49.041,159.146
C08376=1023.219,139.403,387.992,168.063,49.047,159.147
C08377=1023.212,139.120,388.016,168.060,49.052,159.147
C08378=1023.207,138.871,388.036,168.057,49.058,159.148
C08379=1023.201,138.622,388.056,168.054,49.063,159.148
C08380=1023.196,138.373,388.077,168.051,49.068,159.149
C08381=1023.191,138.123,388.097,168.047,49.073,159.150
C08382=1023.185,137.875,388.117,168.044,49.079,159.150
C08383=1023.179,137.626,388.138,168.042,49.083,159.151
C08384=1023.173,137.376,388.158,168.039,49.089,159.151
C08385=1023.168,137.126,388.178,168.035,49.094,159.152
C08386=1023.162,136.877,388.198,168.032,49.100,159.153
C08387=1023.157,136.628,388.219,168.029,49.104,159.153
C08388=1023.151,136.379,388.239,168.026,49.110,159.154
C08389=1023.145,136.130,388.259,168.024,49.115,159.154
C08390=1023.140,135.881,388.280,168.021,49.120,159.155
C08391=1023.134,135.632,388.300,168.017,49.125,159.155
C08392=1023.129,135.383,388.320,168.014,49.131,159.156
C08393=1023.123,135.135,388.340,168.011,49.136,159.156
C08394=1023.118,134.885,388.360,168.008,49.141,159.157
C08395=1023.111,134.635,388.380,168.006,49.147,159.158
C08396=1023.106,134.386,388.401,168.002,49.152,159.158
C08397=1023.100,134.137,388.421,167.999,49.157,159.159
C08398=1023.095,133.888,388.441,167.996,49.162,159.159
C08399=1023.089,133.639,388.461,167.993,49.168,159.160
C08400=1023.084,133.390,388.481,167.990,49.173,159.161
C08401=1023.078,133.141,388.501,167.988,49.178,159.161
C08402=1023.073,132.892,388.522,167.984,49.183,159.162
C08403=1023.067,132.643,388.542,167.981,49.188,159.162
C08404=1023.062,132.393,388.561,167.978,49.193,159.163
C08405=1023.056,132.144,388.581,167.976,49.199,159.164
C08406=1023.050,131.895,388.602,167.972,49.204,159.164
C08407=1023.044,131.646,388.622,167.969,49.209,159.165
C08408=1023.039,131.397,388.642,167.966,49.214,159.165
C08409=1023.033,131.148,388.662,167.963,49.220,159.166
C08410=1023.027,130.899,388.682,167.961,49.224,159.166
C08411=1023.022,130.650,388.702,167.958,49.230,159.167
C08412=1023.017,130.400,388.722,167.954,49.235,159.168
C08413=1023.011,130.151,388.742,167.951,49.241,159.168
C08414=1023.006,129.902,388.761,167.948,49.246,159.169
C08415=1023.000,129.653,388.781,167.946,49.251,159.169
C08416=1022.994,129.404,388.801,167.943,49.256,159.170
C08417=1022.989,129.155,388.821,167.940,49.262,159.171
C08418=1022.983,128.906,388.841,167.937,49.267,159.171
C08419=1022.977,128.656,388.860,167.934,49.273,159.172
C08420=1022.971,128.408,388.880,167.931,49.278,159.172
C08421=1022.965,128.158,388.899,167.928,49.283,159.173
C08422=1022.959,127.909,388.919,167.925,49.288,159.174
C08423=1022.954,127.660,388.939,167.922,49.294,159.174
C08424=1022.948,127.411,388.959,167.919,49.299,159.175
C08425=1022.943,127.161,388.978,167.916,49.305,159.175
C08426=1022.937,126.912,388.998,167.913,49.310,159.176
C08427=1022.931,126.663,389.018,167.910,49.315,159.177
C08428=1022.925,126.414,389.038,167.907,49.321,159.177
C08429=1022.919,126.165,389.057,167.904,49.326,159.178
C08430=1022.914,125.915,389.076,167.901,49.331,159.178
C08431=1022.908,125.666,389.097,167.898,49.337,159.179
C08432=1022.903,125.417,389.116,167.896,49.342,159.180
C08433=1022.897,125.168,389.136,167.893,49.347,159.180
C08434=1022.891,124.919,389.155,167.890,49.353,159.181
C08435=1022.886,124.670,389.175,167.887,49.358,159.182
C08436=1022.880,124.421,389.194,167.883,49.363,159.182
C08437=1022.874,124.172,389.213,167.881,49.369,159.183
C08438=1022.868,123.888,389.236,167.877,49.375,159.183
C08439=1022.861,123.604,389.258,167.875,49.381,159.184
C08440=1022.855,123.321,389.280,167.871,49.387,159.185
C08441=1022.848,123.037,389.303,167.868,49.393,159.185
C08442=1022.843,122.789,389.322,167.865,49.398,159.186
C08443=1022.838,122.539,389.342,167.862,49.404,159.187
C08444=1022.832,122.290,389.361,167.858,49.409,159.187
C08445=1022.826,122.041,389.381,167.856,49.414,159.188
C08446=1022.820,121.791,389.400,167.853,49.420,159.188
C08447=1022.815,121.542,389.420,167.850,49.425,159.189
C08448=1022.809,121.293,389.440,167.847,49.430,159.190
C08449=1022.803,121.044,389.459,167.845,49.435,159.190
C08450=1022.798,120.795,389.478,167.842,49.441,159.191
C08451=1022.792,120.546,389.498,167.839,49.446,159.191
C08452=1022.787,120.296,389.518,167.836,49.451,159.192
C08453=1022.781,120.047,389.537,167.833,49.457,159.193
C08454=1022.775,119.798,389.557,167.830,49.462,159.193
C08455=1022.770,119.549,389.576,167.827,49.467,159.194
C08456=1022.764,119.300,389.595,167.825,49.473,159.194
C08457=1022.759,119.051,389.614,167.822,49.477,159.195
C08458=1022.753,118.802,389.634,167.819,49.483,159.196
C08459=1022.747,118.552,389.653,167.815,49.488,159.196
C08460=1022.742,118.303,389.673,167.814,49.493,159.197
C08461=1022.737,118.054,389.692,167.810,49.498,159.197
C08462=1022.731,117.804,389.711,167.807,49.504,159.198
C08463=1022.725,117.556,389.731,167.805,49.509,159.199
C08464=1022.720,117.306,389.750,167.802,49.514,159.199
C08465=1022.714,117.057,389.770,167.799,49.520,159.200
C08466=1022.709,116.808,389.789,167.796,49.525,159.200
C08467=1022.703,116.559,389.809,167.794,49.530,159.201
C08468=1022.697,116.310,389.828,167.790,49.535,159.201
C08469=1022.692,116.060,389.847,167.787,49.541,159.202
C08470=1022.687,115.811,389.866,167.785,49.546,159.203
C08471=1022.682,115.562,389.886,167.782,49.551,159.203
C08472=1022.676,115.312,389.905,167.779,49.556,159.204
C08473=1022.670,115.064,389.925,167.777,49.562,159.204
C08474=1022.665,114.815,389.944,167.774,49.567,159.205
C08475=1022.659,114.565,389.963,167.770,49.572,159.205
C08476=1022.653,114.316,389.982,167.768,49.578,159.206
C08477=1022.648,114.067,390.002,167.765,49.583,159.207
C08478=1022.643,113.818,390.020,167.762,49.588,159.207
C08479=1022.637,113.568,390.040,167.760,49.593,159.208
C08480=1022.632,113.319,390.059,167.757,49.599,159.209
C08481=1022.627,113.071,390.079,167.754,49.604,159.209
C08482=1022.621,112.821,390.098,167.752,49.609,159.210
C08483=1022.615,112.572,390.118,167.748,49.614,159.210
C08484=1022.609,112.322,390.137,167.745,49.620,159.211
C08485=1022.604,112.074,390.156,167.743,49.624,159.211
C08486=1022.598,111.824,390.174,167.740,49.630,159.212
C08487=1022.593,111.574,390.193,167.737,49.636,159.213
C08488=1022.587,111.325,390.212,167.735,49.640,159.213
C08489=1022.582,111.076,390.231,167.732,49.646,159.214
C08490=1022.576,110.827,390.250,167.729,49.652,159.214
C08491=1022.570,110.578,390.269,167.725,49.657,159.215
C08492=1022.565,110.329,390.288,167.724,49.662,159.216
C08493=1022.559,110.080,390.307,167.721,49.668,159.216
C08494=1022.553,109.830,390.326,167.717,49.673,159.217
C08495=1022.548,109.581,390.345,167.715,49.678,159.218
C08496=1022.542,109.332,390.364,167.712,49.684,159.218
C08497=1022.536,109.082,390.382,167.709,49.689,159.219
C08498=1022.530,108.833,390.401,167.706,49.694,159.219
C08499=1022.525,108.584,390.420,167.704,49.700,159.220
C08500=1022.519,108.335,390.439,167.701,49.705,159.220
C08501=1022.513,108.085,390.457,167.698,49.711,159.221
C08502=1022.507,107.802,390.479,167.695,49.717,159.222
C08503=1022.500,107.518,390.500,167.691,49.723,159.222
C08504=1022.494,107.235,390.521,167.689,49.729,159.223
C08505=1022.487,106.951,390.543,167.686,49.735,159.224
C08506=1022.482,106.701,390.561,167.683,49.741,159.225
C08507=1022.476,106.453,390.580,167.679,49.746,159.225
C08508=1022.470,106.203,390.599,167.677,49.751,159.226
C08509=1022.465,105.954,390.618,167.675,49.757,159.226
C08510=1022.459,105.705,390.636,167.671,49.762,159.227
C08511=1022.453,105.456,390.655,167.668,49.767,159.227
C08512=1022.448,105.207,390.673,167.666,49.773,159.228
C08513=1022.442,104.957,390.692,167.663,49.778,159.229
C08514=1022.436,104.708,390.711,167.660,49.784,159.229
C08515=1022.431,104.459,390.729,167.658,49.789,159.230
C08516=1022.425,104.209,390.748,167.655,49.794,159.231
C08517=1022.420,103.960,390.767,167.652,49.800,159.231
C08518=1022.414,103.711,390.785,167.650,49.805,159.232
C08519=1022.408,103.462,390.805,167.647,49.810,159.232
C08520=1022.403,103.213,390.822,167.644,49.816,159.233
C08521=1022.397,102.963,390.841,167.642,49.821,159.234
C08522=1022.392,102.714,390.860,167.638,49.826,159.234
C08523=1022.386,102.465,390.878,167.636,49.832,159.235
C08524=1022.380,102.215,390.898,167.634,49.837,159.236
C08525=1022.374,101.966,390.915,167.630,49.842,159.236
C08526=1022.369,101.717,390.934,167.627,49.848,159.237
C08527=1022.364,101.468,390.953,167.625,49.853,159.237
C08528=1022.358,101.219,390.971,167.622,49.858,159.238
C08529=1022.352,100.970,390.990,167.619,49.864,159.239
C08530=1022.347,100.720,391.009,167.617,49.869,159.239
C08531=1022.341,100.471,391.027,167.614,49.874,159.240
C08532=1022.336,100.222,391.046,167.611,49.879,159.240
C08533=1022.329,99.972,391.064,167.609,49.885,159.241
C08534=1022.324,99.723,391.083,167.606,49.891,159.242
C08535=1022.319,99.473,391.101,167.602,49.896,159.242
C08536=1022.313,99.225,391.120,167.601,49.901,159.243
C08537=1022.307,98.975,391.138,167.598,49.907,159.243
C08538=1022.302,98.726,391.156,167.594,49.912,159.244
C08539=1022.296,98.477,391.174,167.592,49.917,159.245
C08540=1022.290,98.227,391.192,167.589,49.923,159.245
C08541=1022.285,97.978,391.211,167.587,49.929,159.246
C08542=1022.279,97.729,391.229,167.583,49.934,159.246
C08543=1022.273,97.479,391.247,167.581,49.939,159.247
C08544=1022.267,97.230,391.266,167.578,49.945,159.248
C08545=1022.262,96.981,391.284,167.575,49.950,159.248
C08546=1022.255,96.732,391.302,167.573,49.955,159.249
C08547=1022.251,96.483,391.320,167.570,49.961,159.249
C08548=1022.244,96.233,391.338,167.567,49.967,159.250
C08549=1022.239,95.984,391.357,167.565,49.971,159.251
C08550=1022.233,95.734,391.375,167.562,49.977,159.251
C08551=1022.228,95.485,391.393,167.559,49.983,159.252
C08552=1022.221,95.236,391.411,167.557,49.987,159.253
C08553=1022.216,94.987,391.429,167.554,49.993,159.253
C08554=1022.210,94.737,391.447,167.551,49.999,159.254
C08555=1022.205,94.489,391.466,167.549,50.004,159.254
C08556=1022.198,94.239,391.484,167.546,50.009,159.255
C08557=1022.194,93.990,391.502,167.543,50.015,159.256
C08558=1022.187,93.740,391.520,167.541,50.020,159.256
C08559=1022.182,93.491,391.538,167.538,50.026,159.257
C08560=1022.177,93.242,391.556,167.535,50.031,159.257
C08561=1022.171,92.992,391.574,167.533,50.036,159.258
C08562=1022.165,92.744,391.592,167.530,50.042,159.259
C08563=1022.160,92.494,391.611,167.527,50.047,159.259
C08564=1022.154,92.245,391.629,167.525,50.052,159.260
C08565=1022.148,91.996,391.647,167.522,50.058,159.260
C08566=1022.143,91.776,391.663,167.519,50.063,159.261
C08567=1022.139,91.556,391.679,167.517,50.067,159.262
C08568=1022.134,91.337,391.695,167.515,50.072,159.262
C08569=1022.128,91.116,391.711,167.513,50.077,159.263
C08570=1022.123,90.897,391.727,167.510,50.082,159.263
C08571=1022.118,90.677,391.742,167.507,50.087,159.264
C08572=1022.114,90.457,391.759,167.505,50.091,159.264
C08573=1022.108,90.237,391.775,167.503,50.096,159.265
C08574=1022.103,89.988,391.792,167.500,50.101,159.265
C08575=1022.098,89.739,391.810,167.497,50.107,159.266
C08576=1022.092,89.489,391.828,167.494,50.112,159.266
C08577=1022.086,89.240,391.846,167.492,50.117,159.267
C08578=1022.080,88.990,391.864,167.489,50.123,159.268
C08579=1022.075,88.741,391.881,167.486,50.128,159.268
C08580=1022.069,88.492,391.899,167.484,50.133,159.269
C08581=1022.063,88.242,391.917,167.481,50.139,159.270
C08582=1022.057,87.994,391.935,167.478,50.145,159.270
C08583=1022.051,87.744,391.953,167.476,50.149,159.271
C08584=1022.046,87.495,391.971,167.473,50.155,159.271
C08585=1022.040,87.246,391.988,167.470,50.161,159.272
C08586=1022.034,86.996,392.006,167.468,50.166,159.273
C08587=1022.028,86.747,392.024,167.465,50.171,159.273
C08588=1022.022,86.498,392.042,167.462,50.177,159.274
C08589=1022.017,86.249,392.059,167.459,50.183,159.274
C08590=1022.011,86.000,392.077,167.457,50.188,159.275
C08591=1022.005,85.750,392.095,167.454,50.193,159.276
C08592=1022.000,85.500,392.112,167.451,50.199,159.276
C08593=1021.994,85.251,392.129,167.449,50.205,159.277
C08594=1021.988,85.001,392.147,167.446,50.210,159.277
C08595=1021.983,84.752,392.165,167.443,50.215,159.278
C08596=1021.977,84.503,392.182,167.441,50.221,159.279
C08597=1021.971,84.254,392.200,167.438,50.227,159.280
C08598=1021.966,84.005,392.218,167.435,50.232,159.280
C08599=1021.960,83.756,392.235,167.433,50.237,159.281
C08600=1021.954,83.506,392.253,167.430,50.243,159.281
C08601=1021.948,83.257,392.271,167.427,50.248,159.282
C08602=1021.943,83.008,392.288,167.425,50.253,159.283
C08603=1021.937,82.758,392.306,167.422,50.259,159.283
C08604=1021.931,82.509,392.324,167.420,50.264,159.284
C08605=1021.926,82.260,392.342,167.417,50.270,159.284
C08606=1021.920,82.010,392.359,167.414,50.275,159.285
C08607=1021.914,81.760,392.376,167.412,50.280,159.286
C08608=1021.909,81.511,392.394,167.409,50.286,159.286
C08609=1021.903,81.262,392.411,167.406,50.291,159.287
C08610=1021.897,81.013,392.429,167.404,50.297,159.287
C08611=1021.892,80.764,392.447,167.401,50.302,159.288
C08612=1021.886,80.515,392.464,167.398,50.307,159.288
C08613=1021.880,80.264,392.482,167.396,50.313,159.289
C08614=1021.875,80.015,392.499,167.393,50.319,159.290
C08615=1021.869,79.766,392.517,167.391,50.323,159.290
C08616=1021.864,79.517,392.534,167.388,50.329,159.291
C08617=1021.858,79.267,392.552,167.385,50.334,159.291
C08618=1021.850,78.925,392.575,167.382,50.342,159.292
C08619=1021.842,78.583,392.600,167.378,50.349,159.293
C08620=1021.835,78.240,392.624,167.374,50.356,159.294
C08621=1021.827,77.897,392.648,167.371,50.364,159.295
C08622=1021.822,77.648,392.666,167.369,50.369,159.296
C08623=1021.816,77.399,392.683,167.366,50.374,159.296
C08624=1021.810,77.149,392.700,167.363,50.380,159.297
C08625=1021.804,76.900,392.717,167.360,50.385,159.297
C08626=1021.798,76.651,392.735,167.358,50.391,159.298
C08627=1021.793,76.401,392.752,167.355,50.396,159.298
C08628=1021.788,76.152,392.769,167.353,50.401,159.299
C08629=1021.781,75.903,392.786,167.350,50.407,159.300
C08630=1021.775,75.619,392.806,167.347,50.413,159.300
C08631=1021.769,75.336,392.826,167.343,50.420,159.301
C08632=1021.762,75.052,392.845,167.341,50.426,159.302
C08633=1021.756,74.768,392.865,167.338,50.432,159.302
C08634=1021.749,74.520,392.882,167.335,50.438,159.303
C08635=1021.744,74.270,392.899,167.332,50.443,159.303
C08636=1021.739,74.021,392.916,167.330,50.448,159.304
C08637=1021.732,73.771,392.933,167.327,50.454,159.305
C08638=1021.727,73.522,392.951,167.325,50.459,159.305
C08639=1021.721,73.273,392.968,167.322,50.464,159.306
C08640=1021.715,73.023,392.984,167.319,50.470,159.307
C08641=1021.710,72.774,393.002,167.317,50.475,159.307
C08642=1021.704,72.524,393.019,167.314,50.481,159.308
C08643=1021.698,72.275,393.036,167.311,50.487,159.308
C08644=1021.692,72.026,393.053,167.309,50.491,159.309
C08645=1021.687,71.777,393.071,167.306,50.497,159.310
C08646=1021.682,71.527,393.087,167.303,50.503,159.310
C08647=1021.675,71.278,393.104,167.301,50.508,159.311
C08648=1021.670,71.029,393.121,167.298,50.514,159.311
C08649=1021.664,70.779,393.139,167.296,50.518,159.312
C08650=1021.658,70.529,393.155,167.293,50.524,159.313
C08651=1021.653,70.280,393.173,167.290,50.530,159.313
C08652=1021.647,70.031,393.189,167.288,50.535,159.314
C08653=1021.641,69.782,393.207,167.285,50.541,159.314
C08654=1021.636,69.532,393.224,167.282,50.546,159.315
C08655=1021.630,69.283,393.240,167.280,50.551,159.316
C08656=1021.624,69.034,393.257,167.277,50.557,159.316
C08657=1021.619,68.784,393.275,167.275,50.562,159.317
C08658=1021.612,68.535,393.292,167.272,50.568,159.317
C08659=1021.607,68.285,393.309,167.269,50.573,159.318
C08660=1021.601,68.036,393.325,167.267,50.578,159.319
C08661=1021.596,67.787,393.342,167.264,50.584,159.319
C08662=1021.590,67.537,393.359,167.261,50.590,159.320
C08663=1021.584,67.288,393.375,167.259,50.595,159.320
C08664=1021.578,67.039,393.392,167.256,50.600,159.321
C08665=1021.573,66.789,393.409,167.253,50.605,159.322
C08666=1021.566,66.539,393.426,167.251,50.611,159.322
C08667=1021.561,66.290,393.443,167.248,50.617,159.323
C08668=1021.555,66.041,393.460,167.245,50.622,159.323
C08669=1021.550,65.791,393.477,167.243,50.627,159.324
C08670=1021.544,65.543,393.494,167.240,50.633,159.325
C08671=1021.538,65.293,393.510,167.237,50.638,159.325
C08672=1021.532,65.044,393.527,167.235,50.644,159.326
C08673=1021.527,64.794,393.543,167.233,50.650,159.327
C08674=1021.521,64.545,393.560,167.230,50.654,159.327
C08675=1021.516,64.296,393.577,167.227,50.660,159.328
C08676=1021.510,64.046,393.594,167.224,50.665,159.328
C08677=1021.504,63.797,393.610,167.222,50.671,159.329
C08678=1021.498,63.548,393.627,167.220,50.677,159.329
C08679=1021.492,63.298,393.644,167.216,50.682,159.330
C08680=1021.487,63.048,393.661,167.215,50.687,159.331
C08681=1021.481,62.799,393.677,167.212,50.693,159.331
C08682=1021.475,62.549,393.693,167.208,50.698,159.332
C08683=1021.469,62.300,393.710,167.207,50.704,159.332
C08684=1021.463,62.050,393.726,167.204,50.709,159.333
C08685=1021.457,61.801,393.743,167.201,50.715,159.334
C08686=1021.452,61.552,393.759,167.198,50.721,159.334
C08687=1021.446,61.302,393.775,167.196,50.726,159.335
C08688=1021.440,61.053,393.792,167.193,50.732,159.336
C08689=1021.434,60.804,393.808,167.190,50.738,159.336
C08690=1021.428,60.554,393.824,167.187,50.743,159.337
C08691=1021.423,60.305,393.841,167.185,50.748,159.337
C08692=1021.417,60.055,393.857,167.182,50.754,159.338
C08693=1021.411,59.806,393.873,167.180,50.760,159.339
C08694=1021.403,59.523,393.892,167.177,50.766,159.339
C08695=1021.397,59.239,393.910,167.174,50.772,159.340
C08696=1021.390,58.956,393.930,167.170,50.778,159.341
C08697=1021.384,58.671,393.948,167.168,50.785,159.341
C08698=1021.378,58.422,393.965,167.165,50.790,159.342
C08699=1021.372,58.173,393.981,167.163,50.796,159.343
C08700=1021.366,57.923,393.997,167.160,50.801,159.343
C08701=1021.360,57.674,394.013,167.157,50.807,159.344
C08702=1021.354,57.425,394.030,167.155,50.812,159.344
C08703=1021.348,57.175,394.046,167.152,50.818,159.345
C08704=1021.343,56.927,394.062,167.149,50.824,159.346
C08705=1021.338,56.676,394.078,167.146,50.829,159.346
C08706=1021.332,56.427,394.094,167.144,50.834,159.347
C08707=1021.326,56.178,394.110,167.142,50.840,159.347
C08708=1021.320,55.928,394.127,167.138,50.845,159.348
C08709=1021.314,55.679,394.143,167.137,50.851,159.349
C08710=1021.308,55.430,394.159,167.134,50.857,159.349
C08711=1021.302,55.180,394.175,167.131,50.862,159.350
C08712=1021.296,54.931,394.192,167.129,50.867,159.350
C08713=1021.291,54.681,394.209,167.126,50.873,159.351
C08714=1021.285,54.432,394.225,167.123,50.878,159.351
C08715=1021.279,54.182,394.240,167.121,50.884,159.352
C08716=1021.273,53.933,394.257,167.118,50.889,159.353
C08717=1021.268,53.683,394.273,167.115,50.895,159.353
C08718=1021.262,53.435,394.289,167.113,50.900,159.354
C08719=1021.256,53.185,394.305,167.110,50.906,159.354
C08720=1021.250,52.936,394.321,167.108,50.911,159.355
C08721=1021.245,52.686,394.338,167.105,50.916,159.356
C08722=1021.239,52.436,394.354,167.102,50.922,159.356
C08723=1021.233,52.187,394.370,167.100,50.927,159.357
C08724=1021.227,51.938,394.386,167.097,50.933,159.357
C08725=1021.222,51.688,394.402,167.094,50.938,159.358
C08726=1021.216,51.440,394.418,167.092,50.943,159.359
C08727=1021.211,51.190,394.434,167.089,50.949,159.359
C08728=1021.205,50.940,394.450,167.086,50.954,159.360
C08729=1021.199,50.691,394.466,167.084,50.960,159.360
C08730=1021.193,50.441,394.483,167.081,50.965,159.361
C08731=1021.187,50.192,394.499,167.079,50.971,159.362
C08732=1021.182,49.942,394.515,167.076,50.976,159.362
C08733=1021.176,49.693,394.531,167.073,50.982,159.363
C08734=1021.171,49.444,394.547,167.071,50.987,159.363
C08735=1021.165,49.195,394.563,167.068,50.992,159.364
C08736=1021.159,48.945,394.579,167.065,50.998,159.364
C08737=1021.153,48.695,394.595,167.064,51.003,159.365
C08738=1021.147,48.446,394.611,167.060,51.008,159.365
C08739=1021.143,48.196,394.627,167.059,51.014,159.366
C08740=1021.137,47.947,394.644,167.055,51.019,159.367
C08741=1021.131,47.698,394.660,167.053,51.025,159.367
C08742=1021.125,47.448,394.676,167.050,51.030,159.368
C08743=1021.119,47.198,394.692,167.048,51.035,159.368
C08744=1021.114,46.950,394.707,167.045,51.040,159.369
C08745=1021.108,46.700,394.724,167.042,51.045,159.369
C08746=1021.102,46.450,394.739,167.039,51.051,159.370
C08747=1021.096,46.201,394.756,167.037,51.056,159.371
C08748=1021.091,45.952,394.771,167.034,51.062,159.371
C08749=1021.086,45.702,394.788,167.032,51.067,159.372
C08750=1021.080,45.453,394.804,167.030,51.073,159.372
C08751=1021.074,45.204,394.820,167.027,51.078,159.373
C08752=1021.069,44.954,394.835,167.024,51.083,159.373
C08753=1021.063,44.705,394.851,167.021,51.089,159.374
C08754=1021.057,44.456,394.868,167.019,51.093,159.374
C08755=1021.052,44.206,394.883,167.016,51.099,159.375
C08756=1021.046,43.957,394.899,167.014,51.104,159.376
C08757=1021.041,43.707,394.915,167.011,51.109,159.376
C08758=1021.034,43.423,394.933,167.008,51.115,159.377
C08759=1021.028,43.139,394.952,167.005,51.121,159.377
C08760=1021.022,42.856,394.969,167.003,51.128,159.378
C08761=1021.015,42.572,394.988,166.999,51.134,159.379
C08762=1021.009,42.322,395.003,166.997,51.139,159.379
C08763=1021.004,42.073,395.019,166.994,51.145,159.380
C08764=1020.998,41.823,395.035,166.991,51.150,159.380
C08765=1020.992,41.574,395.051,166.989,51.155,159.381
C08766=1020.987,41.325,395.066,166.986,51.161,159.381
C08767=1020.981,41.076,395.082,166.983,51.166,159.382
C08768=1020.975,40.826,395.097,166.981,51.171,159.383
C08769=1020.969,40.576,395.113,166.978,51.177,159.383
C08770=1020.963,40.327,395.128,166.976,51.182,159.384
C08771=1020.958,40.077,395.144,166.974,51.188,159.384
C08772=1020.952,39.828,395.160,166.970,51.193,159.385
C08773=1020.947,39.579,395.175,166.969,51.199,159.385
C08774=1020.941,39.329,395.191,166.965,51.204,159.386
C08775=1020.934,39.080,395.206,166.963,51.210,159.387
C08776=1020.929,38.831,395.222,166.961,51.215,159.387
C08777=1020.924,38.581,395.237,166.957,51.220,159.388
C08778=1020.918,38.331,395.253,166.955,51.226,159.388
C08779=1020.913,38.082,395.269,166.952,51.231,159.389
C08780=1020.906,37.833,395.284,166.950,51.236,159.389
C08781=1020.900,37.583,395.300,166.948,51.241,159.390
C08782=1020.895,37.334,395.315,166.945,51.247,159.390
C08783=1020.890,37.084,395.331,166.942,51.252,159.391
C08784=1020.884,36.834,395.347,166.939,51.257,159.391
C08785=1020.878,36.585,395.361,166.937,51.263,159.392
C08786=1020.872,36.335,395.377,166.933,51.268,159.392
C08787=1020.867,36.085,395.392,166.932,51.274,159.393
C08788=1020.861,35.837,395.408,166.929,51.280,159.394
C08789=1020.855,35.587,395.423,166.926,51.285,159.394
C08790=1020.849,35.338,395.438,166.924,51.291,159.395
C08791=1020.843,35.088,395.453,166.921,51.296,159.395
C08792=1020.837,34.839,395.468,166.918,51.302,159.396
C08793=1020.831,34.589,395.485,166.916,51.307,159.397
C08794=1020.825,34.340,395.499,166.913,51.312,159.397
C08795=1020.820,34.090,395.515,166.910,51.318,159.398
C08796=1020.815,33.841,395.530,166.908,51.323,159.398
C08797=1020.808,33.591,395.545,166.905,51.328,159.399
C08798=1020.803,33.341,395.560,166.902,51.334,159.399
C08799=1020.797,33.092,395.575,166.900,51.339,159.400
C08800=1020.791,32.843,395.591,166.898,51.345,159.401
C08801=1020.785,32.594,395.606,166.894,51.350,159.401
C08802=1020.779,32.344,395.621,166.893,51.356,159.402
C08803=1020.773,32.095,395.636,166.889,51.361,159.402
C08804=1020.768,31.845,395.651,166.887,51.367,159.403
C08805=1020.762,31.595,395.667,166.885,51.372,159.403
C08806=1020.757,31.346,395.682,166.881,51.377,159.404
C08807=1020.751,31.096,395.697,166.879,51.383,159.404
C08808=1020.745,30.847,395.712,166.877,51.388,159.405
C08809=1020.740,30.597,395.727,166.874,51.394,159.406
C08810=1020.733,30.348,395.742,166.871,51.399,159.406
C08811=1020.728,30.099,395.757,166.869,51.405,159.407
C08812=1020.721,29.850,395.773,166.866,51.410,159.407
C08813=1020.716,29.600,395.788,166.863,51.415,159.408
C08814=1020.710,29.351,395.803,166.861,51.421,159.408
C08815=1020.705,29.101,395.818,166.858,51.426,159.409
C08816=1020.699,28.851,395.834,166.855,51.432,159.409
C08817=1020.694,28.602,395.848,166.853,51.437,159.410
C08818=1020.688,28.352,395.864,166.850,51.442,159.410
C08819=1020.682,28.103,395.879,166.847,51.448,159.411
C08820=1020.676,27.854,395.894,166.845,51.453,159.411
C08821=1020.671,27.605,395.909,166.842,51.458,159.412
C08822=1020.664,27.320,395.926,166.839,51.464,159.413
C08823=1020.657,27.036,395.943,166.837,51.470,159.413
C08824=1020.651,26.752,395.960,166.833,51.477,159.414
C08825=1020.645,26.469,395.977,166.830,51.483,159.414
C08826=1020.638,26.219,395.992,166.827,51.488,159.415
C08827=1020.633,25.970,396.006,166.825,51.493,159.416
C08828=1020.627,25.719,396.021,166.822,51.499,159.416
C08829=1020.621,25.471,396.036,166.819,51.504,159.417
C08830=1020.615,25.221,396.051,166.816,51.510,159.417
C08831=1020.610,24.972,396.066,166.814,51.515,159.418
C08832=1020.604,24.722,396.081,166.811,51.521,159.418
C08833=1020.598,24.473,396.095,166.808,51.526,159.419
C08834=1020.593,24.222,396.110,166.806,51.531,159.419
C08835=1020.587,23.973,396.125,166.804,51.537,159.420
C08836=1020.581,23.725,396.139,166.800,51.542,159.420
C08837=1020.575,23.475,396.154,166.799,51.548,159.421
C08838=1020.570,23.225,396.169,166.796,51.553,159.422
C08839=1020.563,22.975,396.184,166.792,51.559,159.422
C08840=1020.558,22.726,396.198,166.791,51.564,159.423
C08841=1020.552,22.476,396.214,166.788,51.569,159.423
C08842=1020.546,22.227,396.228,166.785,51.575,159.424
C08843=1020.540,21.977,396.243,166.783,51.580,159.424
C08844=1020.534,21.728,396.257,166.780,51.585,159.425
C08845=1020.529,21.479,396.272,166.777,51.591,159.425
C08846=1020.523,21.229,396.287,166.774,51.597,159.426
C08847=1020.517,20.980,396.301,166.772,51.602,159.426
C08848=1020.512,20.730,396.317,166.769,51.607,159.427
C08849=1020.506,20.481,396.331,166.766,51.613,159.427
C08850=1020.501,20.231,396.345,166.764,51.618,159.428
C08851=1020.494,19.982,396.360,166.761,51.624,159.428
C08852=1020.489,19.732,396.375,166.759,51.628,159.429
C08853=1020.483,19.482,396.390,166.756,51.634,159.429
C08854=1020.477,19.233,396.404,166.753,51.640,159.430
C08855=1020.472,18.984,396.419,166.751,51.645,159.431
C08856=1020.466,18.733,396.434,166.748,51.650,159.431
C08857=1020.460,18.485,396.448,166.745,51.656,159.432
C08858=1020.455,18.235,396.462,166.742,51.661,159.432
C08859=1020.449,17.985,396.477,166.740,51.667,159.433
C08860=1020.443,17.736,396.492,166.737,51.672,159.433
C08861=1020.437,17.486,396.506,166.734,51.677,159.434
C08862=1020.431,17.237,396.520,166.732,51.683,159.434
C08863=1020.426,16.987,396.535,166.729,51.688,159.435
C08864=1020.420,16.738,396.550,166.726,51.693,159.435
C08865=1020.414,16.488,396.564,166.724,51.699,159.436
C08866=1020.409,16.239,396.578,166.721,51.704,159.436
C08867=1020.402,15.989,396.593,166.718,51.709,159.437
C08868=1020.397,15.740,396.607,166.715,51.715,159.437
C08869=1020.391,15.491,396.622,166.713,51.720,159.438
C08870=1020.386,15.240,396.636,166.710,51.725,159.438
C08871=1020.380,14.991,396.651,166.707,51.731,159.439
C08872=1020.374,14.742,396.665,166.705,51.736,159.439
C08873=1020.368,14.493,396.679,166.702,51.741,159.440
C08874=1020.362,14.243,396.694,166.699,51.747,159.440
C08875=1020.357,13.994,396.708,166.697,51.752,159.441
C08876=1020.351,13.744,396.722,166.694,51.758,159.441
C08877=1020.345,13.494,396.736,166.692,51.764,159.442
C08878=1020.339,13.245,396.751,166.689,51.768,159.443
C08879=1020.334,12.995,396.765,166.686,51.774,159.443
C08880=1020.327,12.746,396.780,166.684,51.780,159.444
C08881=1020.322,12.496,396.794,166.680,51.785,159.444
C08882=1020.316,12.246,396.807,166.679,51.791,159.445
C08883=1020.311,11.997,396.821,166.676,51.796,159.445
C08884=1020.305,11.747,396.836,166.673,51.802,159.446
C08885=1020.298,11.498,396.850,166.670,51.807,159.446
C08886=1020.292,11.215,396.866,166.667,51.813,159.447
C08887=1020.286,10.934,396.882,166.664,51.819,159.447
C08888=1020.279,10.651,396.898,166.661,51.825,159.448
C08889=1020.272,10.368,396.913,166.658,51.831,159.449
C08890=1020.267,10.119,396.927,166.655,51.837,159.449
C08891=1020.261,9.870,396.942,166.652,51.843,159.450
C08892=1020.255,9.620,396.956,166.650,51.848,159.450
C08893=1020.249,9.370,396.970,166.647,51.853,159.451
C08894=1020.244,9.121,396.984,166.644,51.859,159.451
C08895=1020.237,8.872,396.998,166.642,51.865,159.452
C08896=1020.231,8.622,397.012,166.639,51.870,159.452
C08897=1020.226,8.372,397.026,166.636,51.875,159.453
C08898=1020.220,8.122,397.040,166.634,51.881,159.453
C08899=1020.215,7.873,397.053,166.631,51.886,159.454
C08900=1020.209,7.624,397.068,166.628,51.891,159.454
C08901=1020.202,7.374,397.082,166.626,51.897,159.455
C08902=1020.197,7.124,397.096,166.623,51.902,159.455
C08903=1020.191,6.875,397.109,166.620,51.908,159.456
C08904=1020.186,6.625,397.123,166.618,51.913,159.456
C08905=1020.180,6.376,397.137,166.615,51.918,159.457
C08906=1020.174,6.126,397.152,166.612,51.924,159.457
C08907=1020.168,5.877,397.165,166.610,51.929,159.458
C08908=1020.162,5.627,397.179,166.607,51.935,159.458
C08909=1020.157,5.378,397.193,166.604,51.940,159.459
C08910=1020.151,5.128,397.207,166.601,51.945,159.459
C08911=1020.146,4.878,397.221,166.599,51.950,159.460
C08912=1020.140,4.629,397.234,166.596,51.956,159.460
C08913=1020.133,4.380,397.249,166.593,51.961,159.461
C08914=1020.128,4.130,397.263,166.591,51.966,159.461
C08915=1020.122,3.880,397.277,166.588,51.972,159.462
C08916=1020.117,3.631,397.291,166.585,51.978,159.462
C08917=1020.111,3.381,397.304,166.582,51.983,159.463
C08918=1020.105,3.132,397.318,166.580,51.988,159.463
C08919=1020.100,2.882,397.332,166.577,51.993,159.464
C08920=1020.094,2.633,397.345,166.574,51.998,159.464
C08921=1020.088,2.383,397.360,166.572,52.004,159.465
C08922=1020.083,2.133,397.374,166.569,52.009,159.465
C08923=1020.076,1.884,397.387,166.566,52.015,159.466
C08924=1020.071,1.634,397.401,166.564,52.020,159.466
C08925=1020.065,1.385,397.415,166.561,52.025,159.467
C08926=1020.060,1.135,397.428,166.558,52.031,159.467
C08927=1020.054,0.885,397.442,166.556,52.036,159.468
C08928=1020.049,0.636,397.456,166.553,52.041,159.468
C08929=1020.043,0.387,397.469,166.550,52.046,159.468
C08930=1020.037,0.137,397.483,166.547,52.052,159.469
C08931=1020.032,-0.113,397.497,166.544,52.057,159.469
C08932=1020.026,-0.362,397.511,166.541,52.062,159.470
C08933=1020.021,-0.612,397.525,166.538,52.067,159.470
C08934=1020.015,-0.861,397.538,166.537,52.073,159.471
C08935=1020.009,-1.111,397.552,166.534,52.078,159.471
C08936=1020.003,-1.361,397.566,166.530,52.083,159.472
C08937=1019.998,-1.610,397.580,166.528,52.088,159.472
C08938=1019.992,-1.860,397.594,166.525,52.094,159.473
C08939=1019.986,-2.109,397.607,166.522,52.099,159.473
C08940=1019.980,-2.359,397.621,166.520,52.104,159.474
C08941=1019.975,-2.608,397.635,166.517,52.109,159.474
C08942=1019.969,-2.858,397.649,166.514,52.114,159.474
C08943=1019.964,-3.108,397.663,166.512,52.119,159.475
C08944=1019.958,-3.357,397.676,166.509,52.125,159.475
C08945=1019.952,-3.606,397.690,166.507,52.130,159.476
C08946=1019.947,-3.857,397.703,166.504,52.135,159.476
C08947=1019.942,-4.106,397.717,166.501,52.140,159.477
C08948=1019.935,-4.355,397.730,166.498,52.145,159.477
C08949=1019.930,-4.605,397.744,166.496,52.151,159.478
C08950=1019.924,-4.886,397.759,166.492,52.158,159.478
C08951=1019.917,-5.166,397.773,166.489,52.164,159.479
C08952=1019.911,-5.447,397.789,166.486,52.169,159.479
C08953=1019.903,-5.727,397.804,166.483,52.175,159.480
C08954=1019.898,-5.977,397.817,166.480,52.181,159.480
C08955=1019.892,-6.226,397.830,166.478,52.186,159.481
C08956=1019.887,-6.476,397.844,166.475,52.192,159.481
C08957=1019.881,-6.726,397.856,166.472,52.197,159.482
C08958=1019.875,-6.975,397.870,166.469,52.202,159.482
C08959=1019.870,-7.224,397.883,166.467,52.208,159.483
C08960=1019.864,-7.474,397.896,166.464,52.213,159.483
C08961=1019.858,-7.723,397.910,166.461,52.218,159.484
C08962=1019.852,-7.972,397.923,166.458,52.224,159.484
C08963=1019.847,-8.223,397.936,166.456,52.229,159.485
C08964=1019.841,-8.472,397.949,166.453,52.235,159.485
C08965=1019.835,-8.722,397.962,166.450,52.240,159.486
C08966=1019.829,-8.971,397.976,166.447,52.245,159.486
C08967=1019.824,-9.221,397.990,166.445,52.250,159.487
C08968=1019.818,-9.471,398.002,166.442,52.256,159.487
C08969=1019.812,-9.720,398.015,166.439,52.261,159.487
C08970=1019.806,-9.970,398.029,166.436,52.266,159.488
C08971=1019.801,-10.219,398.041,166.434,52.272,159.489
C08972=1019.796,-10.469,398.055,166.431,52.277,159.489
C08973=1019.789,-10.718,398.068,166.428,52.283,159.489
C08974=1019.784,-10.968,398.082,166.425,52.288,159.490
C08975=1019.778,-11.218,398.094,166.423,52.293,159.490
C08976=1019.772,-11.467,398.108,166.420,52.298,159.491
C08977=1019.767,-11.717,398.121,166.417,52.304,159.491
C08978=1019.760,-11.966,398.134,166.414,52.309,159.491
C08979=1019.756,-12.216,398.147,166.412,52.314,159.492
C08980=1019.750,-12.465,398.160,166.408,52.319,159.492
C08981=1019.745,-12.715,398.173,166.405,52.324,159.493
C08982=1019.738,-12.965,398.186,166.403,52.331,159.493
C08983=1019.732,-13.215,398.199,166.401,52.335,159.494
C08984=1019.727,-13.464,398.213,166.398,52.341,159.494
C08985=1019.722,-13.713,398.225,166.395,52.346,159.495
C08986=1019.716,-13.963,398.239,166.393,52.351,159.495
C08987=1019.710,-14.213,398.251,166.389,52.356,159.496
C08988=1019.704,-14.463,398.264,166.386,52.362,159.496
C08989=1019.699,-14.712,398.278,166.383,52.367,159.496
C08990=1019.694,-14.961,398.290,166.381,52.372,159.497
C08991=1019.688,-15.211,398.304,166.378,52.377,159.497
C08992=1019.682,-15.461,398.316,166.375,52.383,159.498
C08993=1019.676,-15.710,398.330,166.373,52.388,159.498
C08994=1019.671,-15.960,398.343,166.370,52.393,159.499
C08995=1019.665,-16.209,398.355,166.367,52.398,159.499
C08996=1019.660,-16.459,398.368,166.364,52.404,159.499
C08997=1019.653,-16.709,398.381,166.361,52.409,159.500
C08998=1019.647,-16.959,398.393,166.359,52.414,159.500
C08999=1019.642,-17.209,398.407,166.356,52.419,159.501
C09000=1019.637,-17.457,398.420,166.353,52.425,159.501
C09001=1019.631,-17.707,398.432,166.350,52.431,159.502
C09002=1019.625,-17.957,398.445,166.347,52.436,159.502
C09003=1019.619,-18.207,398.457,166.345,52.441,159.503
C09004=1019.614,-18.456,398.469,166.342,52.446,159.503
C09005=1019.607,-18.705,398.483,166.339,52.452,159.503
C09006=1019.602,-18.956,398.496,166.336,52.457,159.504
C09007=1019.596,-19.205,398.508,166.334,52.462,159.504
C09008=1019.591,-19.455,398.521,166.331,52.467,159.505
C09009=1019.585,-19.705,398.533,166.328,52.473,159.505
C09010=1019.579,-19.954,398.546,166.325,52.479,159.506
C09011=1019.574,-20.203,398.559,166.322,52.484,159.506
C09012=1019.568,-20.453,398.571,166.320,52.489,159.507
C09013=1019.562,-20.703,398.584,166.317,52.494,159.507
C09014=1019.556,-20.981,398.598,166.314,52.500,159.507
C09015=1019.550,-21.259,398.612,166.310,52.506,159.508
C09016=1019.543,-21.539,398.627,166.307,52.512,159.509
C09017=1019.537,-21.817,398.640,166.304,52.518,159.509
C09018=1019.531,-22.067,398.653,166.301,52.523,159.509
C09019=1019.525,-22.316,398.665,166.298,52.528,159.510
C09020=1019.520,-22.566,398.678,166.295,52.534,159.510
C09021=1019.514,-22.816,398.691,166.293,52.539,159.511
C09022=1019.509,-23.065,398.703,166.290,52.544,159.511
C09023=1019.503,-23.315,398.716,166.287,52.549,159.511
C09024=1019.497,-23.565,398.729,166.284,52.555,159.512
C09025=1019.492,-23.814,398.741,166.281,52.560,159.512
C09026=1019.486,-24.064,398.754,166.279,52.565,159.513
C09027=1019.480,-24.314,398.766,166.276,52.570,159.513
C09028=1019.475,-24.563,398.779,166.273,52.576,159.514
C09029=1019.469,-24.813,398.791,166.271,52.581,159.514
C09030=1019.464,-25.062,398.804,166.268,52.586,159.514
C09031=1019.458,-25.312,398.816,166.265,52.591,159.515
C09032=1019.452,-25.562,398.829,166.262,52.597,159.515
C09033=1019.447,-25.811,398.841,166.260,52.602,159.516
C09034=1019.441,-26.061,398.853,166.256,52.606,159.516
C09035=1019.436,-26.310,398.866,166.253,52.612,159.516
C09036=1019.430,-26.560,398.878,166.250,52.617,159.517
C09037=1019.425,-26.810,398.891,166.248,52.622,159.517
C09038=1019.419,-27.059,398.904,166.245,52.628,159.518
C09039=1019.413,-27.309,398.916,166.242,52.633,159.518
C09040=1019.408,-27.558,398.928,166.239,52.638,159.518
C09041=1019.402,-27.808,398.941,166.237,52.643,159.519
C09042=1019.397,-28.059,398.953,166.234,52.649,159.519
C09043=1019.391,-28.308,398.965,166.231,52.654,159.520
C09044=1019.385,-28.558,398.977,166.228,52.659,159.520
C09045=1019.379,-28.807,398.989,166.225,52.665,159.520
C09046=1019.373,-29.057,399.002,166.223,52.670,159.521
C09047=1019.368,-29.306,399.014,166.220,52.675,159.521
C09048=1019.363,-29.556,399.026,166.217,52.680,159.522
C09049=1019.357,-29.806,399.038,166.214,52.686,159.522
C09050=1019.351,-30.055,399.050,166.211,52.691,159.523
C09051=1019.345,-30.305,399.062,166.208,52.697,159.523
C09052=1019.340,-30.555,399.074,166.206,52.702,159.523
C09053=1019.334,-30.805,399.086,166.203,52.707,159.524
C09054=1019.328,-31.054,399.098,166.200,52.712,159.524
C09055=1019.323,-31.304,399.111,166.197,52.718,159.525
C09056=1019.317,-31.553,399.122,166.193,52.723,159.525
C09057=1019.311,-31.803,399.134,166.191,52.728,159.526
C09058=1019.306,-32.052,399.147,166.188,52.733,159.526
C09059=1019.300,-32.302,399.159,166.185,52.739,159.526
C09060=1019.295,-32.552,399.171,166.182,52.744,159.527
C09061=1019.289,-32.802,399.183,166.179,52.749,159.527
C09062=1019.283,-33.051,399.195,166.177,52.755,159.528
C09063=1019.277,-33.301,399.207,166.174,52.760,159.528
C09064=1019.272,-33.550,399.219,166.171,52.765,159.528
C09065=1019.266,-33.800,399.231,166.168,52.771,159.529
C09066=1019.261,-34.050,399.243,166.165,52.775,159.529
C09067=1019.255,-34.299,399.254,166.163,52.780,159.529
C09068=1019.249,-34.549,399.267,166.160,52.786,159.530
C09069=1019.244,-34.799,399.278,166.157,52.791,159.530
C09070=1019.238,-35.049,399.291,166.154,52.796,159.531
C09071=1019.233,-35.298,399.303,166.151,52.802,159.531
C09072=1019.228,-35.548,399.315,166.149,52.807,159.531
C09073=1019.221,-35.797,399.327,166.146,52.812,159.532
C09074=1019.216,-36.047,399.338,166.143,52.818,159.532
C09075=1019.210,-36.297,399.351,166.140,52.823,159.533
C09076=1019.205,-36.546,399.363,166.136,52.828,159.533
C09077=1019.200,-36.796,399.374,166.134,52.833,159.533
C09078=1019.193,-37.074,399.388,166.130,52.839,159.534
C09079=1019.187,-37.352,399.401,166.127,52.845,159.534
C09080=1019.181,-37.629,399.414,166.124,52.850,159.535
C09081=1019.175,-37.908,399.427,166.121,52.856,159.535
C09082=1019.169,-38.157,399.440,166.119,52.861,159.536
C09083=1019.163,-38.406,399.451,166.116,52.867,159.536
C09084=1019.158,-38.656,399.463,166.112,52.871,159.536
C09085=1019.152,-38.905,399.475,166.109,52.877,159.536
C09086=1019.147,-39.155,399.487,166.107,52.882,159.537
C09087=1019.141,-39.405,399.499,166.104,52.887,159.537
C09088=1019.136,-39.655,399.510,166.101,52.893,159.538
C09089=1019.131,-39.904,399.522,166.098,52.898,159.538
C09090=1019.124,-40.154,399.534,166.095,52.903,159.539
C09091=1019.119,-40.404,399.545,166.092,52.909,159.539
C09092=1019.113,-40.653,399.556,166.089,52.914,159.539
C09093=1019.107,-40.903,399.568,166.087,52.919,159.540
C09094=1019.102,-41.153,399.579,166.084,52.925,159.540
C09095=1019.097,-41.402,399.591,166.081,52.930,159.541
C09096=1019.090,-41.652,399.603,166.078,52.935,159.541
C09097=1019.085,-41.902,399.614,166.075,52.941,159.541
C09098=1019.079,-42.151,399.625,166.072,52.946,159.542
C09099=1019.073,-42.401,399.638,166.069,52.951,159.542
C09100=1019.068,-42.651,399.649,166.066,52.956,159.542
C09101=1019.063,-42.900,399.660,166.064,52.961,159.543
